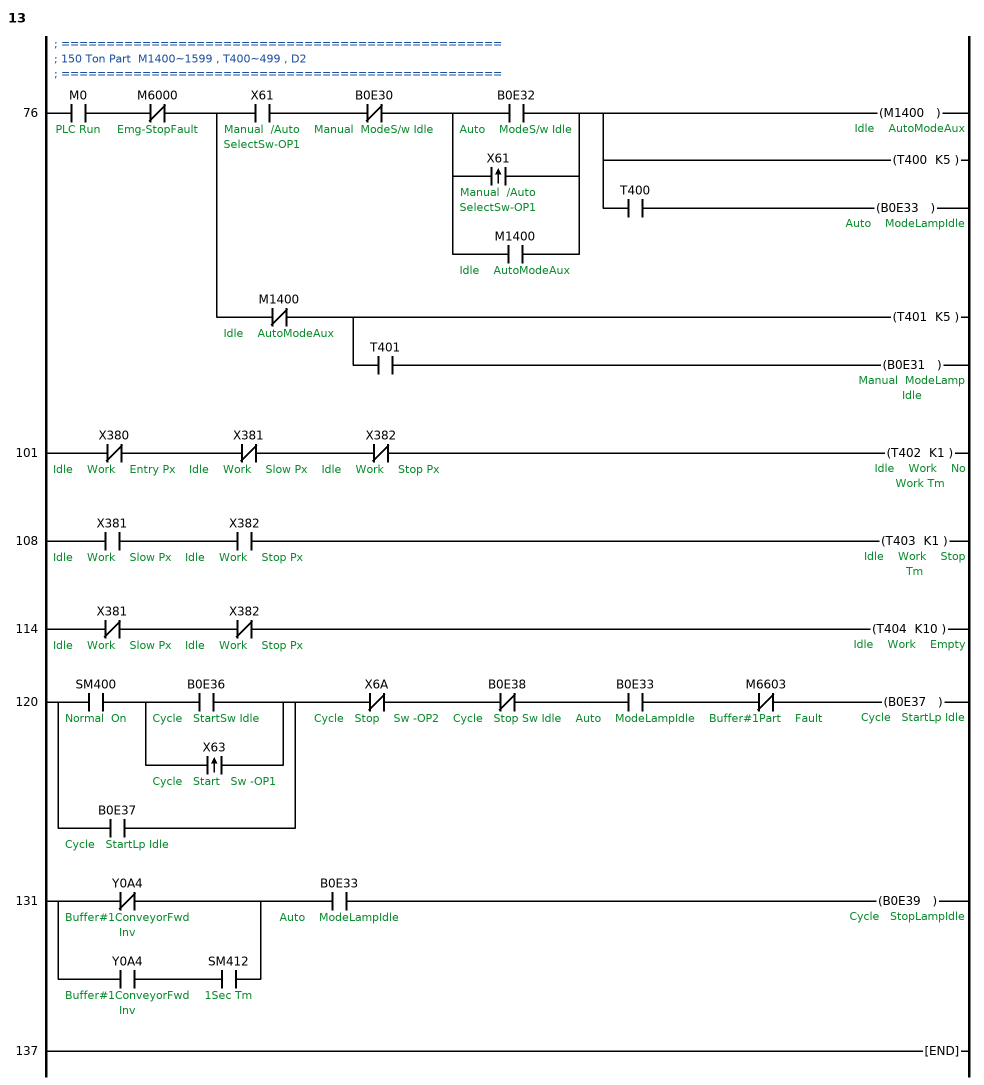
; =================================================
; 150 Ton Part  M1400~1599 , T400~499 , D2
; =================================================
76    LD      M0  ; PLC Run
      ANI     M6000  ; Emg-StopFault
      MPS
      AND     X61  ; Manual  /Auto   SelectSw-OP1
      ANI     B0E30  ; Manual  ModeS/w Idle
      LD      B0E32  ; Auto    ModeS/w Idle
      ORP     X61  ; Manual  /Auto   SelectSw-OP1
      OR      M1400  ; Idle    AutoModeAux
      ANB
      OUT     M1400  ; Idle    AutoModeAux
      OUT     T400 K5
      AND     T400
      OUT     B0E33  ; Auto    ModeLampIdle
      MPP
      ANI     M1400  ; Idle    AutoModeAux
      OUT     T401 K5
      AND     T401
      OUT     B0E31  ; Manual  ModeLampIdle
101   LDI     X380  ; Idle    Work    Entry Px
      ANI     X381  ; Idle    Work    Slow Px
      ANI     X382  ; Idle    Work    Stop Px
      OUT     T402 K1  ; Idle    Work    No Work Tm
108   LD      X381  ; Idle    Work    Slow Px
      AND     X382  ; Idle    Work    Stop Px
      OUT     T403 K1  ; Idle    Work    Stop Tm
114   LDI     X381  ; Idle    Work    Slow Px
      ANI     X382  ; Idle    Work    Stop Px
      OUT     T404 K10  ; Idle    Work    Empty
120   LD      SM400  ; Normal  On
      LD      B0E36  ; Cycle   StartSw Idle
      ORP     X63  ; Cycle   Start   Sw -OP1
      ANB
      OR      B0E37  ; Cycle   StartLp Idle
      ANI     X6A  ; Cycle   Stop    Sw -OP2
      ANI     B0E38  ; Cycle   Stop Sw Idle
      AND     B0E33  ; Auto    ModeLampIdle
      ANI     M6603  ; Buffer#1Part    Fault
      OUT     B0E37  ; Cycle   StartLp Idle
131   LDI     Y0A4  ; Buffer#1ConveyorFwd Inv
      LD      Y0A4  ; Buffer#1ConveyorFwd Inv
      AND     SM412  ; 1Sec Tm
      ORB
      AND     B0E33  ; Auto    ModeLampIdle
      OUT     B0E39  ; Cycle   StopLampIdle
137   END
END_PROGRAM

PROGRAM 14  // Turn Over
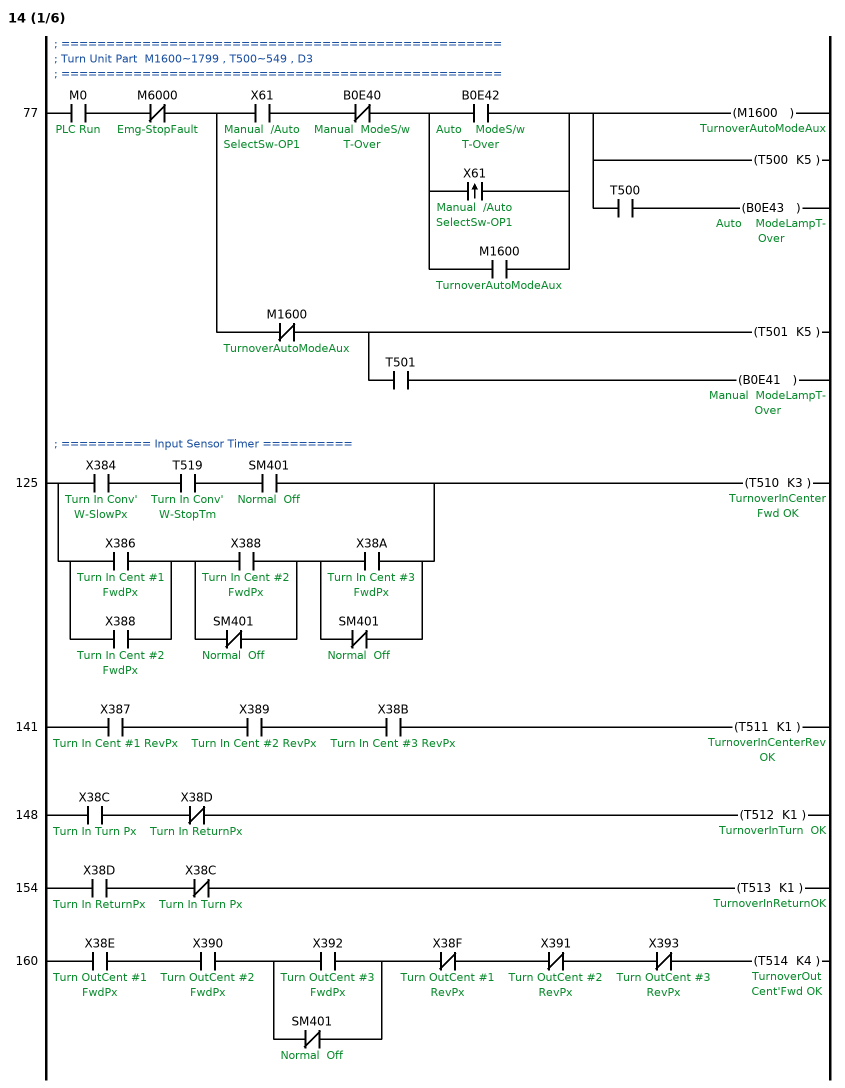
; =================================================
; Turn Unit Part  M1600~1799 , T500~549 , D3
; =================================================
77    LD      M0  ; PLC Run
      ANI     M6000  ; Emg-StopFault
      MPS
      AND     X61  ; Manual  /Auto   SelectSw-OP1
      ANI     B0E40  ; Manual  ModeS/w T-Over
      LD      B0E42  ; Auto    ModeS/w T-Over
      ORP     X61  ; Manual  /Auto   SelectSw-OP1
      OR      M1600  ; TurnoverAutoModeAux
      ANB
      OUT     M1600  ; TurnoverAutoModeAux
      OUT     T500 K5
      AND     T500
      OUT     B0E43  ; Auto    ModeLampT-Over
      MPP
      ANI     M1600  ; TurnoverAutoModeAux
      OUT     T501 K5
      AND     T501
      OUT     B0E41  ; Manual  ModeLampT-Over
; ========== Input Sensor Timer ==========
125   LD      X384  ; Turn In Conv'   W-SlowPx
      AND     T519  ; Turn In Conv'   W-StopTm
      AND     SM401  ; Normal  Off
      LD      X386  ; Turn In Cent #1 FwdPx
      OR      X388  ; Turn In Cent #2 FwdPx
      LD      X388  ; Turn In Cent #2 FwdPx
      ORI     SM401  ; Normal  Off
      ANB
      LD      X38A  ; Turn In Cent #3 FwdPx
      ORI     SM401  ; Normal  Off
      ANB
      ORB
      OUT     T510 K3  ; TurnoverInCenterFwd OK
141   LD      X387  ; Turn In Cent #1 RevPx
      AND     X389  ; Turn In Cent #2 RevPx
      AND     X38B  ; Turn In Cent #3 RevPx
      OUT     T511 K1  ; TurnoverInCenterRev OK
148   LD      X38C  ; Turn In Turn Px
      ANI     X38D  ; Turn In ReturnPx
      OUT     T512 K1  ; TurnoverInTurn  OK
154   LD      X38D  ; Turn In ReturnPx
      ANI     X38C  ; Turn In Turn Px
      OUT     T513 K1  ; TurnoverInReturnOK
160   LD      X38E  ; Turn OutCent #1 FwdPx
      AND     X390  ; Turn OutCent #2 FwdPx
      LD      X392  ; Turn OutCent #3 FwdPx
      ORI     SM401  ; Normal  Off
      ANB
      ANI     X38F  ; Turn OutCent #1 RevPx
      ANI     X391  ; Turn OutCent #2 RevPx
      ANI     X393  ; Turn OutCent #3 RevPx
      OUT     T514 K4  ; TurnoverOutCent'Fwd OK
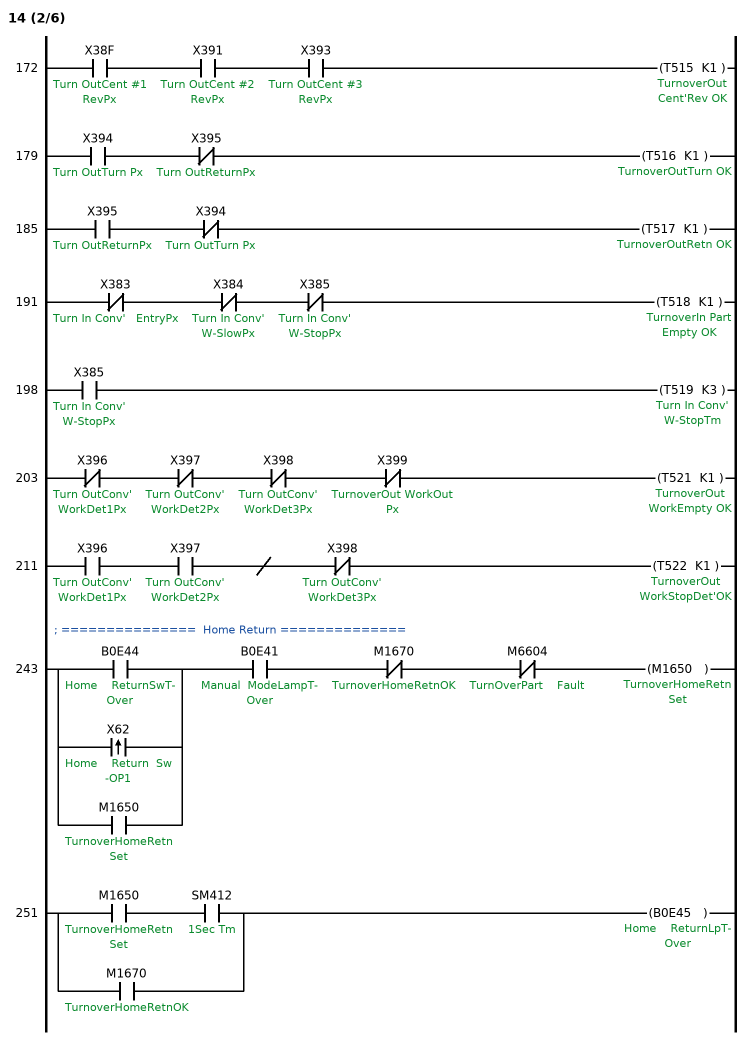
172   LD      X38F  ; Turn OutCent #1 RevPx
      AND     X391  ; Turn OutCent #2 RevPx
      AND     X393  ; Turn OutCent #3 RevPx
      OUT     T515 K1  ; TurnoverOutCent'Rev OK
179   LD      X394  ; Turn OutTurn Px
      ANI     X395  ; Turn OutReturnPx
      OUT     T516 K1  ; TurnoverOutTurn OK
185   LD      X395  ; Turn OutReturnPx
      ANI     X394  ; Turn OutTurn Px
      OUT     T517 K1  ; TurnoverOutRetn OK
191   LDI     X383  ; Turn In Conv'   EntryPx
      ANI     X384  ; Turn In Conv'   W-SlowPx
      ANI     X385  ; Turn In Conv'   W-StopPx
      OUT     T518 K1  ; TurnoverIn Part Empty OK
198   LD      X385  ; Turn In Conv'   W-StopPx
      OUT     T519 K3  ; Turn In Conv'   W-StopTm
203   LDI     X396  ; Turn OutConv'   WorkDet1Px
      ANI     X397  ; Turn OutConv'   WorkDet2Px
      ANI     X398  ; Turn OutConv'   WorkDet3Px
      ANI     X399  ; TurnoverOut WorkOut Px
      OUT     T521 K1  ; TurnoverOut WorkEmpty OK
211   LD      X396  ; Turn OutConv'   WorkDet1Px
      AND     X397  ; Turn OutConv'   WorkDet2Px
      INV
      ANI     X398  ; Turn OutConv'   WorkDet3Px
      OUT     T522 K1  ; TurnoverOut WorkStopDet'OK
; ===============  Home Return ==============
243   LD      B0E44  ; Home    ReturnSwT-Over
      ORP     X62  ; Home    Return  Sw -OP1
      OR      M1650  ; TurnoverHomeRetnSet
      AND     B0E41  ; Manual  ModeLampT-Over
      ANI     M1670  ; TurnoverHomeRetnOK
      ANI     M6604  ; TurnOverPart    Fault
      OUT     M1650  ; TurnoverHomeRetnSet
251   LD      M1650  ; TurnoverHomeRetnSet
      AND     SM412  ; 1Sec Tm
      OR      M1670  ; TurnoverHomeRetnOK
      OUT     B0E45  ; Home    ReturnLpT-Over
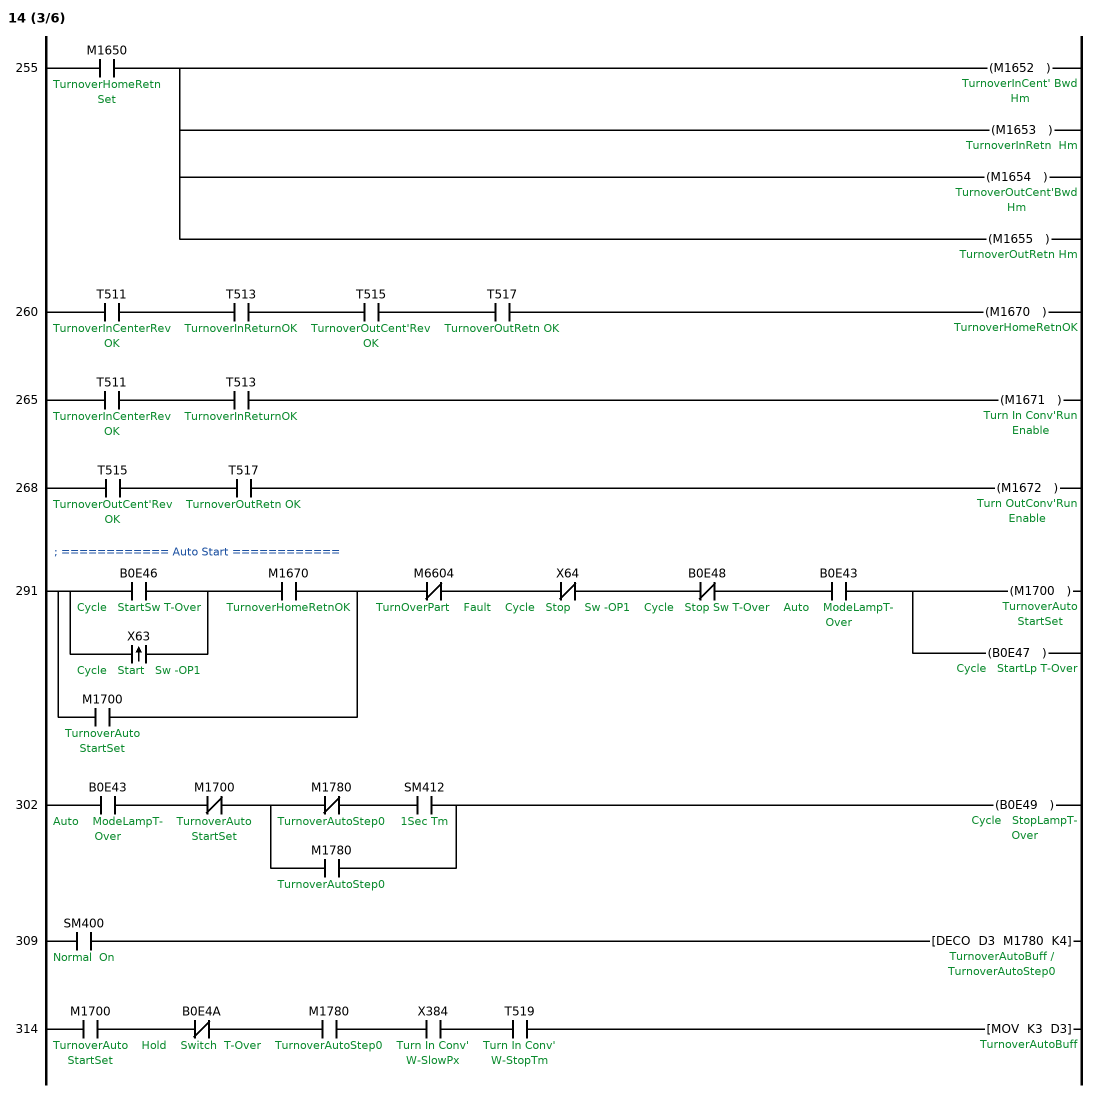
255   LD      M1650  ; TurnoverHomeRetnSet
      OUT     M1652  ; TurnoverInCent' Bwd Hm
      OUT     M1653  ; TurnoverInRetn  Hm
      OUT     M1654  ; TurnoverOutCent'BwdHm
      OUT     M1655  ; TurnoverOutRetn Hm
260   LD      T511  ; TurnoverInCenterRev OK
      AND     T513  ; TurnoverInReturnOK
      AND     T515  ; TurnoverOutCent'Rev OK
      AND     T517  ; TurnoverOutRetn OK
      OUT     M1670  ; TurnoverHomeRetnOK
265   LD      T511  ; TurnoverInCenterRev OK
      AND     T513  ; TurnoverInReturnOK
      OUT     M1671  ; Turn In Conv'RunEnable
268   LD      T515  ; TurnoverOutCent'Rev OK
      AND     T517  ; TurnoverOutRetn OK
      OUT     M1672  ; Turn OutConv'RunEnable
; ============ Auto Start ============
291   LD      B0E46  ; Cycle   StartSw T-Over
      ORP     X63  ; Cycle   Start   Sw -OP1
      AND     M1670  ; TurnoverHomeRetnOK
      OR      M1700  ; TurnoverAuto    StartSet
      ANI     M6604  ; TurnOverPart    Fault
      ANI     X64  ; Cycle   Stop    Sw -OP1
      ANI     B0E48  ; Cycle   Stop Sw T-Over
      AND     B0E43  ; Auto    ModeLampT-Over
      OUT     M1700  ; TurnoverAuto    StartSet
      OUT     B0E47  ; Cycle   StartLp T-Over
302   LD      B0E43  ; Auto    ModeLampT-Over
      ANI     M1700  ; TurnoverAuto    StartSet
      LDI     M1780  ; TurnoverAutoStep0
      AND     SM412  ; 1Sec Tm
      OR      M1780  ; TurnoverAutoStep0
      ANB
      OUT     B0E49  ; Cycle   StopLampT-Over
309   LD      SM400  ; Normal  On
      DECO    D3 M1780 K4  ; TurnoverAutoBuff
314   LD      M1700  ; TurnoverAuto    StartSet
      ANI     B0E4A  ; Hold    Switch  T-Over
      AND     M1780  ; TurnoverAutoStep0
      AND     X384  ; Turn In Conv'   W-SlowPx
      AND     T519  ; Turn In Conv'   W-StopTm
      MOV     K3 D3
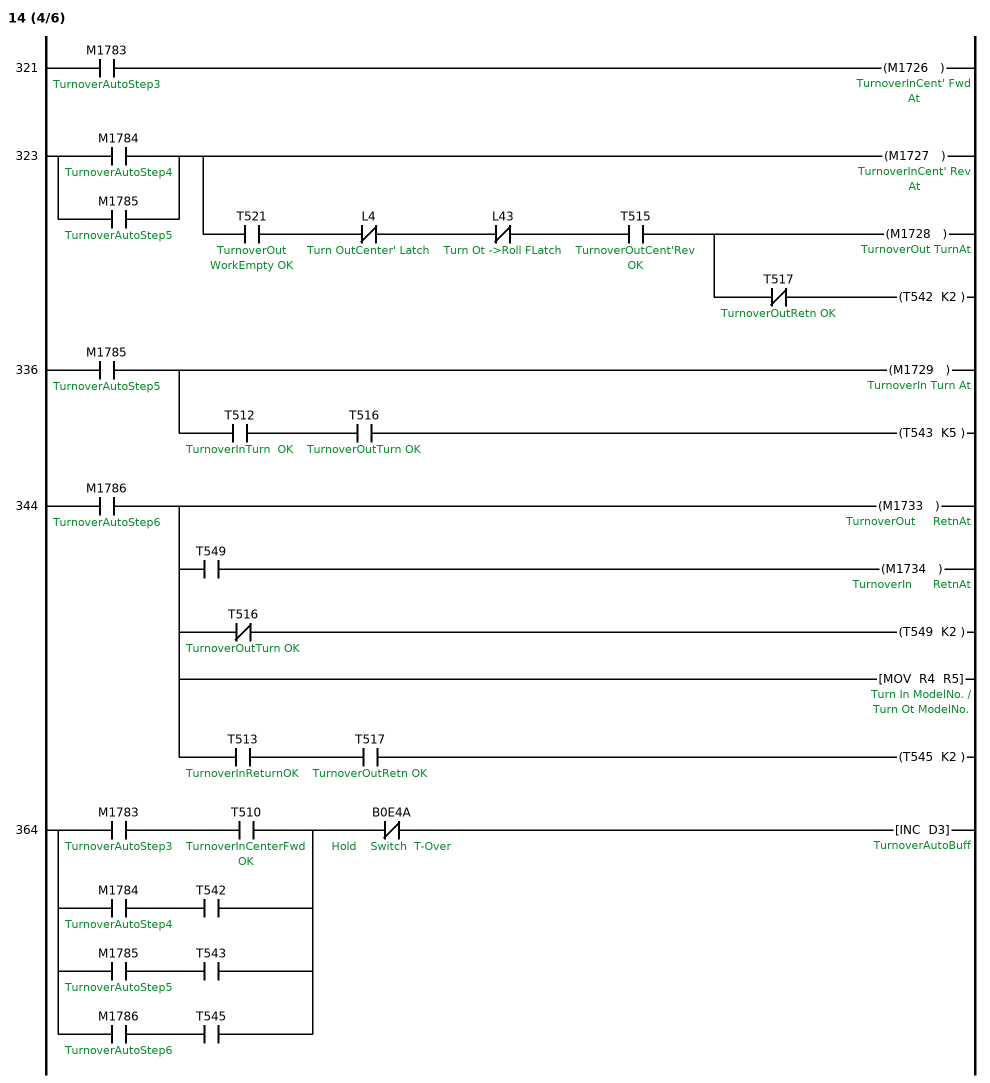
321   LD      M1783  ; TurnoverAutoStep3
      OUT     M1726  ; TurnoverInCent' Fwd At
323   LD      M1784  ; TurnoverAutoStep4
      OR      M1785  ; TurnoverAutoStep5
      OUT     M1727  ; TurnoverInCent' Rev At
      AND     T521  ; TurnoverOut WorkEmpty OK
      ANI     L4  ; Turn OutCenter' Latch
      ANI     L43  ; Turn Ot ->Roll FLatch
      AND     T515  ; TurnoverOutCent'Rev OK
      OUT     M1728  ; TurnoverOut TurnAt
      ANI     T517  ; TurnoverOutRetn OK
      OUT     T542 K2
336   LD      M1785  ; TurnoverAutoStep5
      OUT     M1729  ; TurnoverIn Turn At
      AND     T512  ; TurnoverInTurn  OK
      AND     T516  ; TurnoverOutTurn OK
      OUT     T543 K5
344   LD      M1786  ; TurnoverAutoStep6
      OUT     M1733  ; TurnoverOut     RetnAt
      MPS
      AND     T549
      OUT     M1734  ; TurnoverIn      RetnAt
      MRD
      ANI     T516  ; TurnoverOutTurn OK
      OUT     T549 K2
      MPP
      MOV     R4 R5  ; Turn In ModelNo. / Turn Ot ModelNo.
      AND     T513  ; TurnoverInReturnOK
      AND     T517  ; TurnoverOutRetn OK
      OUT     T545 K2
364   LD      M1783  ; TurnoverAutoStep3
      AND     T510  ; TurnoverInCenterFwd OK
      LD      M1784  ; TurnoverAutoStep4
      AND     T542
      ORB
      LD      M1785  ; TurnoverAutoStep5
      AND     T543
      ORB
      LD      M1786  ; TurnoverAutoStep6
      AND     T545
      ORB
      ANI     B0E4A  ; Hold    Switch  T-Over
      INC     D3
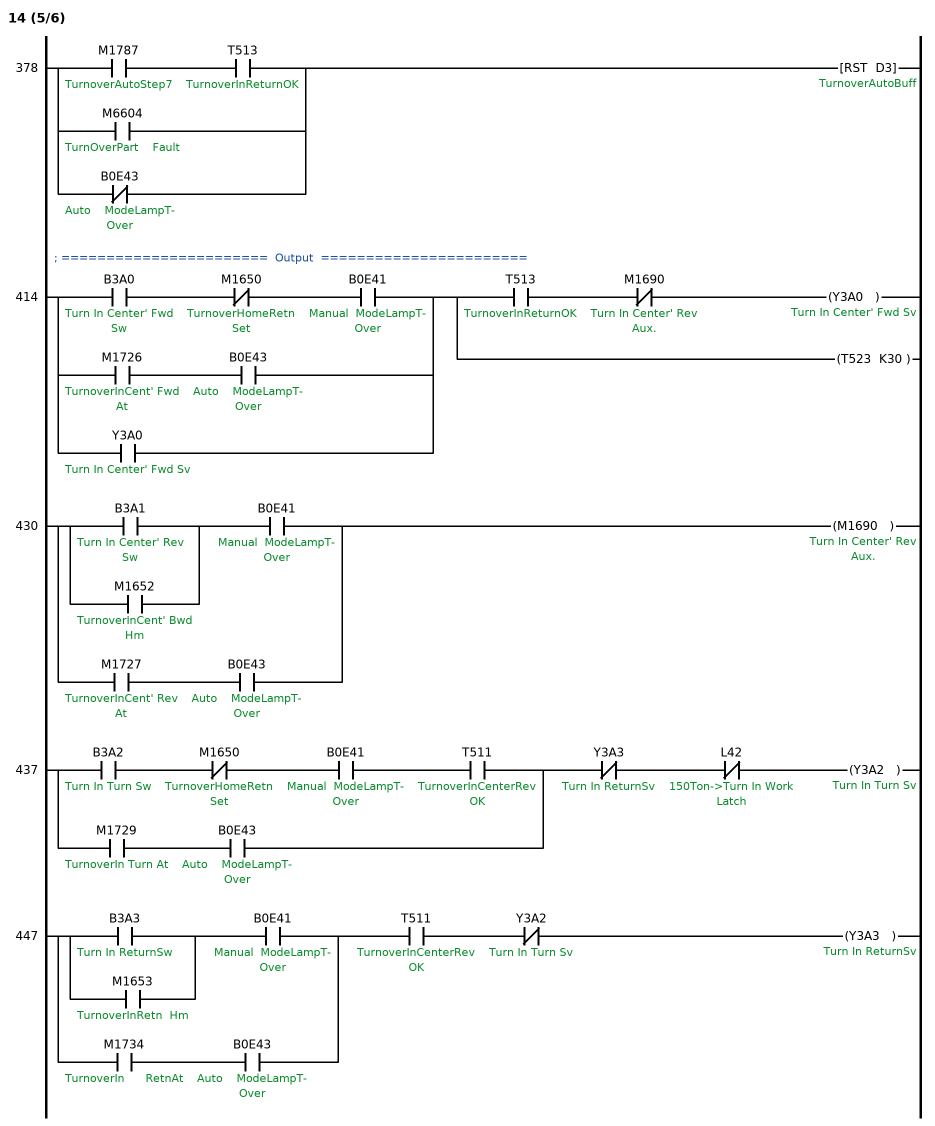
378   LD      M1787  ; TurnoverAutoStep7
      AND     T513  ; TurnoverInReturnOK
      OR      M6604  ; TurnOverPart    Fault
      ORI     B0E43  ; Auto    ModeLampT-Over
      RST     D3  ; TurnoverAutoBuff
; =======================  Output  =======================
414   LD      B3A0  ; Turn In Center' Fwd Sw
      ANI     M1650  ; TurnoverHomeRetnSet
      AND     B0E41  ; Manual  ModeLampT-Over
      LD      M1726  ; TurnoverInCent' Fwd At
      AND     B0E43  ; Auto    ModeLampT-Over
      ORB
      OR      Y3A0  ; Turn In Center' Fwd Sv
      MPS
      AND     T513  ; TurnoverInReturnOK
      ANI     M1690  ; Turn In Center' Rev Aux.
      OUT     Y3A0  ; Turn In Center' Fwd Sv
      MPP
      OUT     T523 K30
430   LD      B3A1  ; Turn In Center' Rev Sw
      OR      M1652  ; TurnoverInCent' Bwd Hm
      AND     B0E41  ; Manual  ModeLampT-Over
      LD      M1727  ; TurnoverInCent' Rev At
      AND     B0E43  ; Auto    ModeLampT-Over
      ORB
      OUT     M1690  ; Turn In Center' Rev Aux.
437   LD      B3A2  ; Turn In Turn Sw
      ANI     M1650  ; TurnoverHomeRetnSet
      AND     B0E41  ; Manual  ModeLampT-Over
      AND     T511  ; TurnoverInCenterRev OK
      LD      M1729  ; TurnoverIn Turn At
      AND     B0E43  ; Auto    ModeLampT-Over
      ORB
      ANI     Y3A3  ; Turn In ReturnSv
      ANI     L42  ; 150Ton->Turn In Work    Latch
      OUT     Y3A2  ; Turn In Turn Sv
447   LD      B3A3  ; Turn In ReturnSw
      OR      M1653  ; TurnoverInRetn  Hm
      AND     B0E41  ; Manual  ModeLampT-Over
      LD      M1734  ; TurnoverIn      RetnAt
      AND     B0E43  ; Auto    ModeLampT-Over
      ORB
      AND     T511  ; TurnoverInCenterRev OK
      ANI     Y3A2  ; Turn In Turn Sv
      OUT     Y3A3  ; Turn In ReturnSv
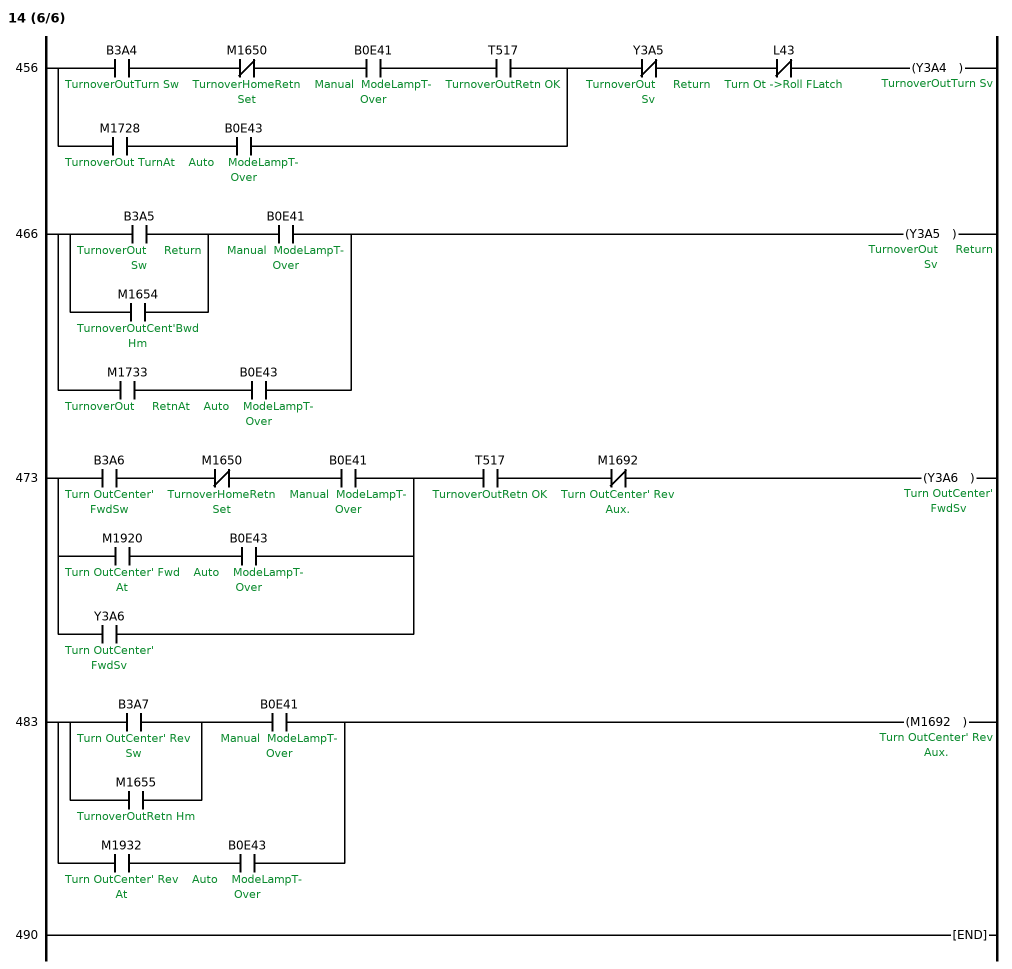
456   LD      B3A4  ; TurnoverOutTurn Sw
      ANI     M1650  ; TurnoverHomeRetnSet
      AND     B0E41  ; Manual  ModeLampT-Over
      AND     T517  ; TurnoverOutRetn OK
      LD      M1728  ; TurnoverOut TurnAt
      AND     B0E43  ; Auto    ModeLampT-Over
      ORB
      ANI     Y3A5  ; TurnoverOut     Return  Sv
      ANI     L43  ; Turn Ot ->Roll FLatch
      OUT     Y3A4  ; TurnoverOutTurn Sv
466   LD      B3A5  ; TurnoverOut     Return  Sw
      OR      M1654  ; TurnoverOutCent'BwdHm
      AND     B0E41  ; Manual  ModeLampT-Over
      LD      M1733  ; TurnoverOut     RetnAt
      AND     B0E43  ; Auto    ModeLampT-Over
      ORB
      OUT     Y3A5  ; TurnoverOut     Return  Sv
473   LD      B3A6  ; Turn OutCenter' FwdSw
      ANI     M1650  ; TurnoverHomeRetnSet
      AND     B0E41  ; Manual  ModeLampT-Over
      LD      M1920  ; Turn OutCenter' Fwd At
      AND     B0E43  ; Auto    ModeLampT-Over
      ORB
      OR      Y3A6  ; Turn OutCenter' FwdSv
      AND     T517  ; TurnoverOutRetn OK
      ANI     M1692  ; Turn OutCenter' Rev Aux.
      OUT     Y3A6  ; Turn OutCenter' FwdSv
483   LD      B3A7  ; Turn OutCenter' Rev Sw
      OR      M1655  ; TurnoverOutRetn Hm
      AND     B0E41  ; Manual  ModeLampT-Over
      LD      M1932  ; Turn OutCenter' Rev At
      AND     B0E43  ; Auto    ModeLampT-Over
      ORB
      OUT     M1692  ; Turn OutCenter' Rev Aux.
490   END
END_PROGRAM

PROGRAM 15  // Roll Forming
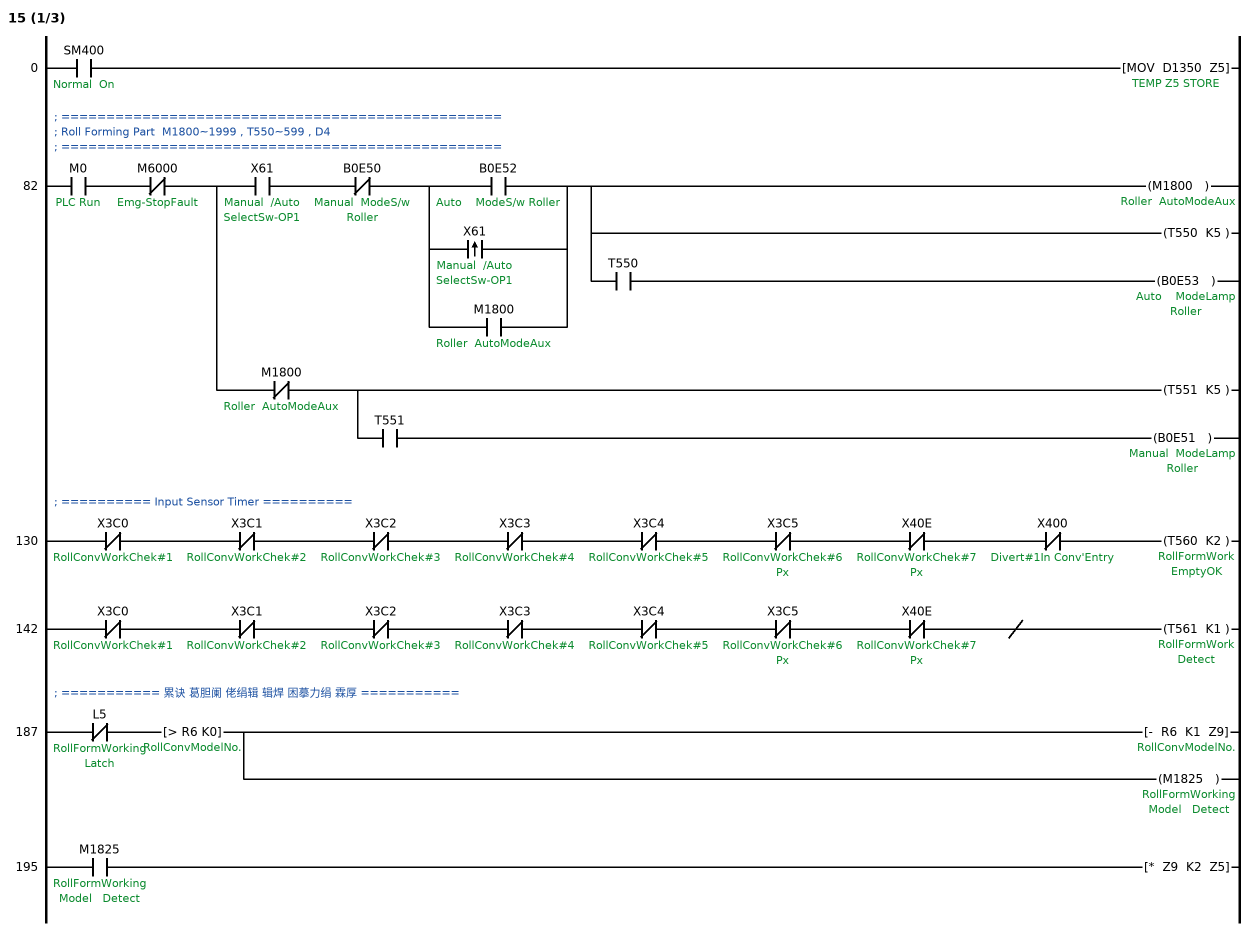
0     LD      SM400  ; Normal  On
      MOV     D1350 Z5  ; TEMP Z5 STORE
; =================================================
; Roll Forming Part  M1800~1999 , T550~599 , D4
; =================================================
82    LD      M0  ; PLC Run
      ANI     M6000  ; Emg-StopFault
      MPS
      AND     X61  ; Manual  /Auto   SelectSw-OP1
      ANI     B0E50  ; Manual  ModeS/w Roller
      LD      B0E52  ; Auto    ModeS/w Roller
      ORP     X61  ; Manual  /Auto   SelectSw-OP1
      OR      M1800  ; Roller  AutoModeAux
      ANB
      OUT     M1800  ; Roller  AutoModeAux
      OUT     T550 K5
      AND     T550
      OUT     B0E53  ; Auto    ModeLampRoller
      MPP
      ANI     M1800  ; Roller  AutoModeAux
      OUT     T551 K5
      AND     T551
      OUT     B0E51  ; Manual  ModeLampRoller
; ========== Input Sensor Timer ==========
130   LDI     X3C0  ; RollConvWorkChek#1
      ANI     X3C1  ; RollConvWorkChek#2
      ANI     X3C2  ; RollConvWorkChek#3
      ANI     X3C3  ; RollConvWorkChek#4
      ANI     X3C4  ; RollConvWorkChek#5
      ANI     X3C5  ; RollConvWorkChek#6 Px
      ANI     X40E  ; RollConvWorkChek#7 Px
      ANI     X400  ; Divert#1In Conv'Entry
      OUT     T560 K2  ; RollFormWork    EmptyOK
142   LDI     X3C0  ; RollConvWorkChek#1
      ANI     X3C1  ; RollConvWorkChek#2
      ANI     X3C2  ; RollConvWorkChek#3
      ANI     X3C3  ; RollConvWorkChek#4
      ANI     X3C4  ; RollConvWorkChek#5
      ANI     X3C5  ; RollConvWorkChek#6 Px
      ANI     X40E  ; RollConvWorkChek#7 Px
      INV
      OUT     T561 K1  ; RollFormWork    Detect
; =========== 작업 모델을 읽어서 서보 위치제어 준비 ===========
187   LDI     L5  ; RollFormWorking Latch
      AND>    R6 K0  ; RollConvModelNo.
      -       R6 K1 Z9
      OUT     M1825  ; RollFormWorking Model   Detect
195   LD      M1825  ; RollFormWorking Model   Detect
      *       Z9 K2 Z5
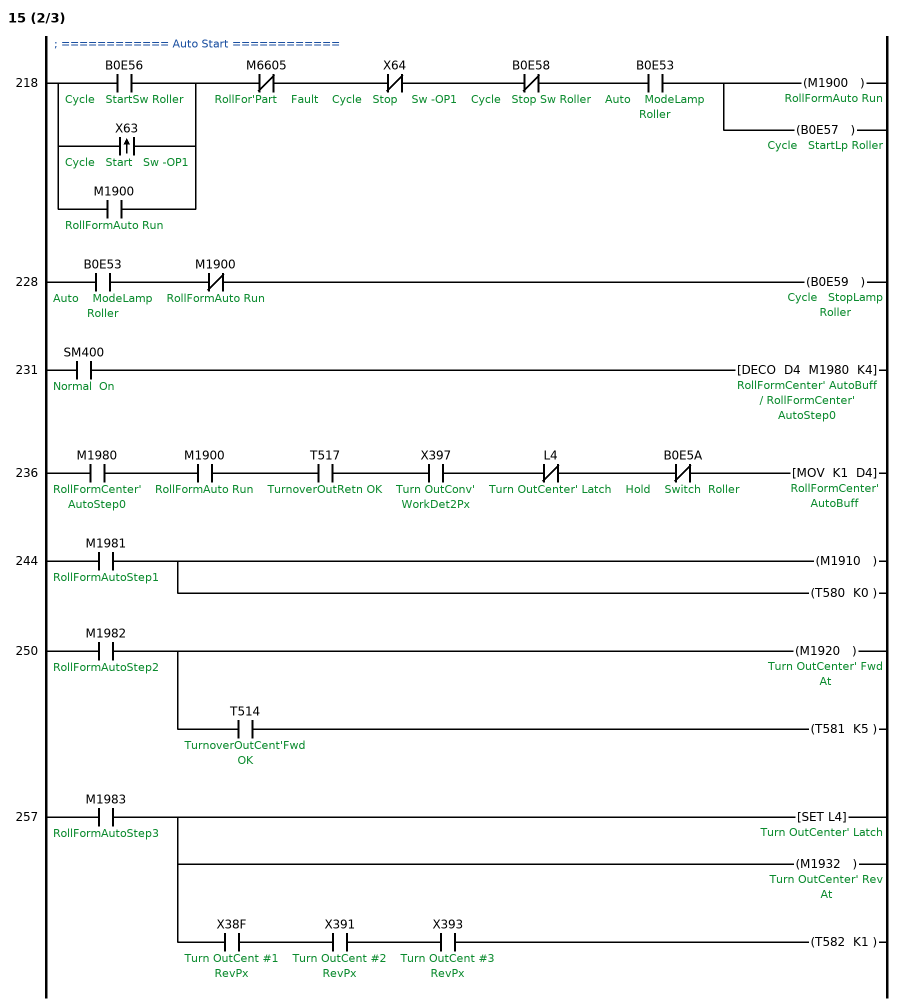
; ============ Auto Start ============
218   LD      B0E56  ; Cycle   StartSw Roller
      ORP     X63  ; Cycle   Start   Sw -OP1
      OR      M1900  ; RollFormAuto Run
      ANI     M6605  ; RollFor'Part    Fault
      ANI     X64  ; Cycle   Stop    Sw -OP1
      ANI     B0E58  ; Cycle   Stop Sw Roller
      AND     B0E53  ; Auto    ModeLampRoller
      OUT     M1900  ; RollFormAuto Run
      OUT     B0E57  ; Cycle   StartLp Roller
228   LD      B0E53  ; Auto    ModeLampRoller
      ANI     M1900  ; RollFormAuto Run
      OUT     B0E59  ; Cycle   StopLampRoller
231   LD      SM400  ; Normal  On
      DECO    D4 M1980 K4  ; RollFormCenter' AutoBuff / RollFormCenter' AutoStep0
236   LD      M1980  ; RollFormCenter' AutoStep0
      AND     M1900  ; RollFormAuto Run
      AND     T517  ; TurnoverOutRetn OK
      AND     X397  ; Turn OutConv'   WorkDet2Px
      ANI     L4  ; Turn OutCenter' Latch
      ANI     B0E5A  ; Hold    Switch  Roller
      MOV     K1 D4
244   LD      M1981  ; RollFormAutoStep1
      OUT     M1910
      OUT     T580 K0
250   LD      M1982  ; RollFormAutoStep2
      OUT     M1920  ; Turn OutCenter' Fwd At
      AND     T514  ; TurnoverOutCent'Fwd OK
      OUT     T581 K5
257   LD      M1983  ; RollFormAutoStep3
      SET     L4  ; Turn OutCenter' Latch
      OUT     M1932  ; Turn OutCenter' Rev At
      AND     X38F  ; Turn OutCent #1 RevPx
      AND     X391  ; Turn OutCent #2 RevPx
      AND     X393  ; Turn OutCent #3 RevPx
      OUT     T582 K1
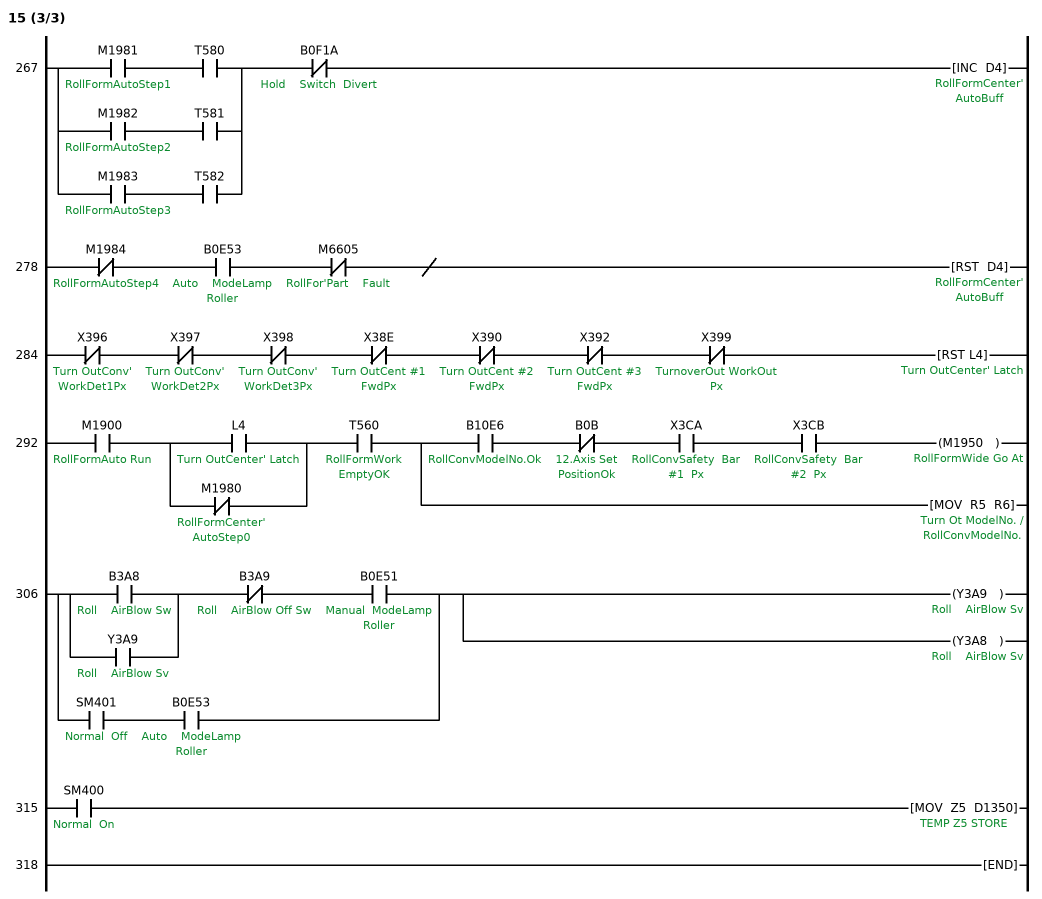
267   LD      M1981  ; RollFormAutoStep1
      AND     T580
      LD      M1982  ; RollFormAutoStep2
      AND     T581
      ORB
      LD      M1983  ; RollFormAutoStep3
      AND     T582
      ORB
      ANI     B0F1A  ; Hold    Switch  Divert
      INC     D4
278   LDI     M1984  ; RollFormAutoStep4
      AND     B0E53  ; Auto    ModeLampRoller
      ANI     M6605  ; RollFor'Part    Fault
      INV
      RST     D4  ; RollFormCenter' AutoBuff
284   LDI     X396  ; Turn OutConv'   WorkDet1Px
      ANI     X397  ; Turn OutConv'   WorkDet2Px
      ANI     X398  ; Turn OutConv'   WorkDet3Px
      ANI     X38E  ; Turn OutCent #1 FwdPx
      ANI     X390  ; Turn OutCent #2 FwdPx
      ANI     X392  ; Turn OutCent #3 FwdPx
      ANI     X399  ; TurnoverOut WorkOut Px
      RST     L4  ; Turn OutCenter' Latch
292   LD      M1900  ; RollFormAuto Run
      LD      L4  ; Turn OutCenter' Latch
      ORI     M1980  ; RollFormCenter' AutoStep0
      ANB
      AND     T560  ; RollFormWork    EmptyOK
      MPS
      AND     B10E6  ; RollConvModelNo.Ok
      ANI     B0B  ; 12.Axis Set     PositionOk
      AND     X3CA  ; RollConvSafety  Bar #1  Px
      AND     X3CB  ; RollConvSafety  Bar #2  Px
      OUT     M1950  ; RollFormWide Go At
      MPP
      MOV     R5 R6  ; Turn Ot ModelNo.
306   LD      B3A8  ; Roll    AirBlow Sw
      OR      Y3A9  ; Roll    AirBlow Sv
      ANI     B3A9  ; Roll    AirBlow Off Sw
      AND     B0E51  ; Manual  ModeLampRoller
      LD      SM401  ; Normal  Off
      AND     B0E53  ; Auto    ModeLampRoller
      ORB
      OUT     Y3A9  ; Roll    AirBlow Sv
      OUT     Y3A8  ; Roll    AirBlow Sv
315   LD      SM400  ; Normal  On
      MOV     Z5 D1350
318   END
END_PROGRAM

PROGRAM 19  // #2 Part Alarm
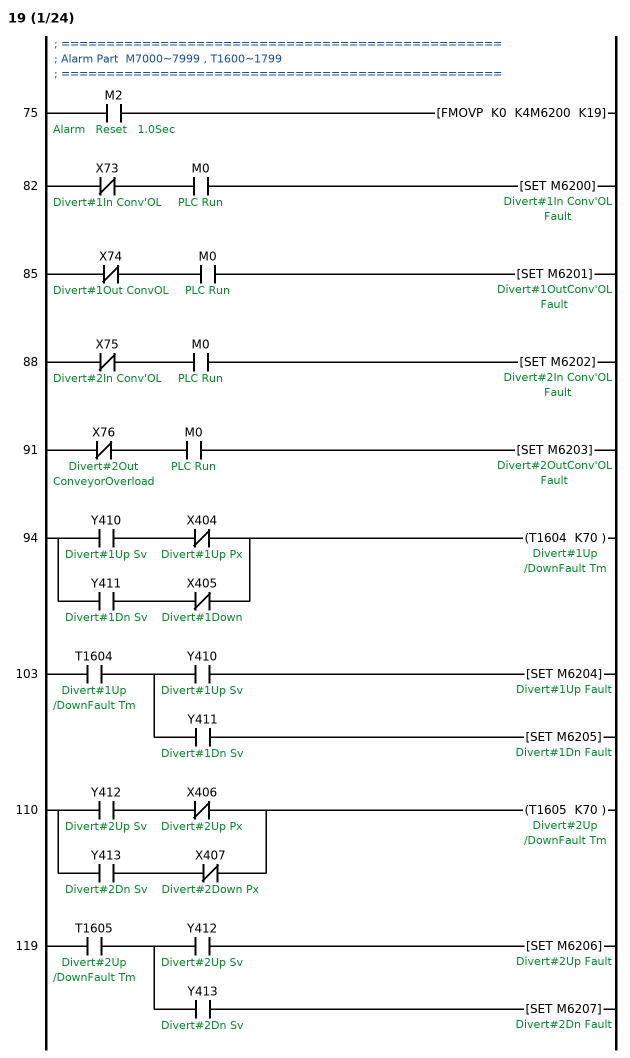
; =================================================
; Alarm Part  M7000~7999 , T1600~1799
; =================================================
75    LD      M2  ; Alarm   Reset   1.0Sec
      FMOVP   K0 K4M6200 K19  ; Divert#1In Conv'OL Fault
82    LDI     X73  ; Divert#1In Conv'OL
      AND     M0  ; PLC Run
      SET     M6200  ; Divert#1In Conv'OL Fault
85    LDI     X74  ; Divert#1Out ConvOL
      AND     M0  ; PLC Run
      SET     M6201  ; Divert#1OutConv'OL Fault
88    LDI     X75  ; Divert#2In Conv'OL
      AND     M0  ; PLC Run
      SET     M6202  ; Divert#2In Conv'OL Fault
91    LDI     X76  ; Divert#2Out     ConveyorOverload
      AND     M0  ; PLC Run
      SET     M6203  ; Divert#2OutConv'OL Fault
94    LD      Y410  ; Divert#1Up Sv
      ANI     X404  ; Divert#1Up Px
      LD      Y411  ; Divert#1Dn Sv
      ANI     X405  ; Divert#1Down
      ORB
      OUT     T1604 K70  ; Divert#1Up /DownFault Tm
103   LD      T1604  ; Divert#1Up /DownFault Tm
      MPS
      AND     Y410  ; Divert#1Up Sv
      SET     M6204  ; Divert#1Up Fault
      MPP
      AND     Y411  ; Divert#1Dn Sv
      SET     M6205  ; Divert#1Dn Fault
110   LD      Y412  ; Divert#2Up Sv
      ANI     X406  ; Divert#2Up Px
      LD      Y413  ; Divert#2Dn Sv
      ANI     X407  ; Divert#2Down Px
      ORB
      OUT     T1605 K70  ; Divert#2Up /DownFault Tm
119   LD      T1605  ; Divert#2Up /DownFault Tm
      MPS
      AND     Y412  ; Divert#2Up Sv
      SET     M6206  ; Divert#2Up Fault
      MPP
      AND     Y413  ; Divert#2Dn Sv
      SET     M6207  ; Divert#2Dn Fault
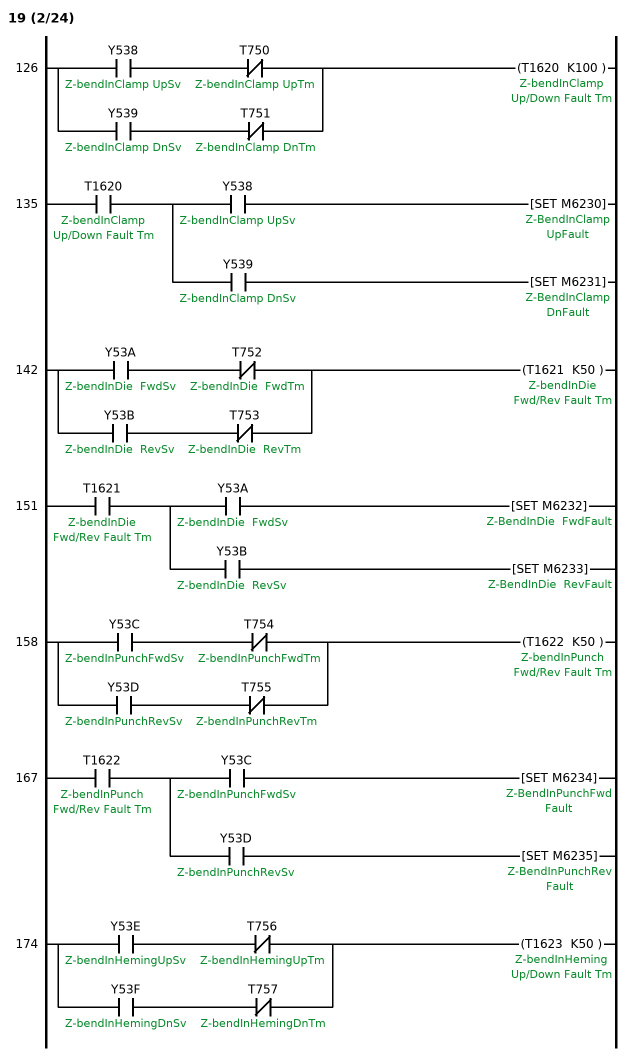
126   LD      Y538  ; Z-bendInClamp UpSv
      ANI     T750  ; Z-bendInClamp UpTm
      LD      Y539  ; Z-bendInClamp DnSv
      ANI     T751  ; Z-bendInClamp DnTm
      ORB
      OUT     T1620 K100  ; Z-bendInClamp   Up/Down Fault Tm
135   LD      T1620  ; Z-bendInClamp   Up/Down Fault Tm
      MPS
      AND     Y538  ; Z-bendInClamp UpSv
      SET     M6230  ; Z-BendInClamp UpFault
      MPP
      AND     Y539  ; Z-bendInClamp DnSv
      SET     M6231  ; Z-BendInClamp DnFault
142   LD      Y53A  ; Z-bendInDie  FwdSv
      ANI     T752  ; Z-bendInDie  FwdTm
      LD      Y53B  ; Z-bendInDie  RevSv
      ANI     T753  ; Z-bendInDie  RevTm
      ORB
      OUT     T1621 K50  ; Z-bendInDie     Fwd/Rev Fault Tm
151   LD      T1621  ; Z-bendInDie     Fwd/Rev Fault Tm
      MPS
      AND     Y53A  ; Z-bendInDie  FwdSv
      SET     M6232  ; Z-BendInDie  FwdFault
      MPP
      AND     Y53B  ; Z-bendInDie  RevSv
      SET     M6233  ; Z-BendInDie  RevFault
158   LD      Y53C  ; Z-bendInPunchFwdSv
      ANI     T754  ; Z-bendInPunchFwdTm
      LD      Y53D  ; Z-bendInPunchRevSv
      ANI     T755  ; Z-bendInPunchRevTm
      ORB
      OUT     T1622 K50  ; Z-bendInPunch   Fwd/Rev Fault Tm
167   LD      T1622  ; Z-bendInPunch   Fwd/Rev Fault Tm
      MPS
      AND     Y53C  ; Z-bendInPunchFwdSv
      SET     M6234  ; Z-BendInPunchFwdFault
      MPP
      AND     Y53D  ; Z-bendInPunchRevSv
      SET     M6235  ; Z-BendInPunchRevFault
174   LD      Y53E  ; Z-bendInHemingUpSv
      ANI     T756  ; Z-bendInHemingUpTm
      LD      Y53F  ; Z-bendInHemingDnSv
      ANI     T757  ; Z-bendInHemingDnTm
      ORB
      OUT     T1623 K50  ; Z-bendInHeming  Up/Down Fault Tm
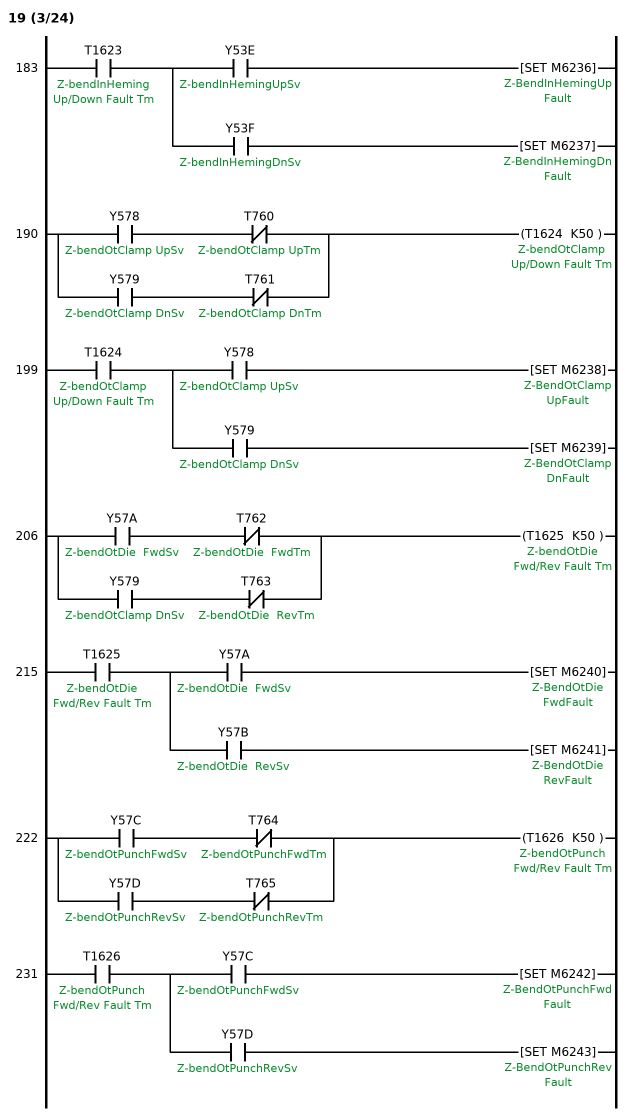
183   LD      T1623  ; Z-bendInHeming  Up/Down Fault Tm
      MPS
      AND     Y53E  ; Z-bendInHemingUpSv
      SET     M6236  ; Z-BendInHemingUpFault
      MPP
      AND     Y53F  ; Z-bendInHemingDnSv
      SET     M6237  ; Z-BendInHemingDnFault
190   LD      Y578  ; Z-bendOtClamp UpSv
      ANI     T760  ; Z-bendOtClamp UpTm
      LD      Y579  ; Z-bendOtClamp DnSv
      ANI     T761  ; Z-bendOtClamp DnTm
      ORB
      OUT     T1624 K50  ; Z-bendOtClamp   Up/Down Fault Tm
199   LD      T1624  ; Z-bendOtClamp   Up/Down Fault Tm
      MPS
      AND     Y578  ; Z-bendOtClamp UpSv
      SET     M6238  ; Z-BendOtClamp UpFault
      MPP
      AND     Y579  ; Z-bendOtClamp DnSv
      SET     M6239  ; Z-BendOtClamp DnFault
206   LD      Y57A  ; Z-bendOtDie  FwdSv
      ANI     T762  ; Z-bendOtDie  FwdTm
      LD      Y579  ; Z-bendOtClamp DnSv
      ANI     T763  ; Z-bendOtDie  RevTm
      ORB
      OUT     T1625 K50  ; Z-bendOtDie     Fwd/Rev Fault Tm
215   LD      T1625  ; Z-bendOtDie     Fwd/Rev Fault Tm
      MPS
      AND     Y57A  ; Z-bendOtDie  FwdSv
      SET     M6240  ; Z-BendOtDie  FwdFault
      MPP
      AND     Y57B  ; Z-bendOtDie  RevSv
      SET     M6241  ; Z-BendOtDie  RevFault
222   LD      Y57C  ; Z-bendOtPunchFwdSv
      ANI     T764  ; Z-bendOtPunchFwdTm
      LD      Y57D  ; Z-bendOtPunchRevSv
      ANI     T765  ; Z-bendOtPunchRevTm
      ORB
      OUT     T1626 K50  ; Z-bendOtPunch   Fwd/Rev Fault Tm
231   LD      T1626  ; Z-bendOtPunch   Fwd/Rev Fault Tm
      MPS
      AND     Y57C  ; Z-bendOtPunchFwdSv
      SET     M6242  ; Z-BendOtPunchFwdFault
      MPP
      AND     Y57D  ; Z-bendOtPunchRevSv
      SET     M6243  ; Z-BendOtPunchRevFault
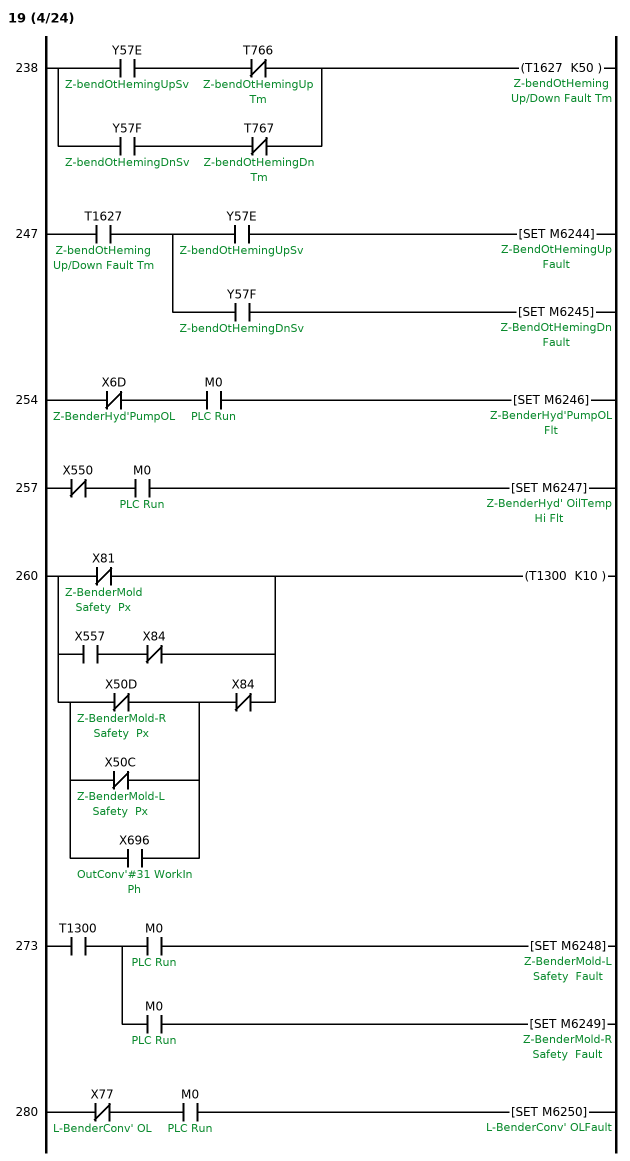
238   LD      Y57E  ; Z-bendOtHemingUpSv
      ANI     T766  ; Z-bendOtHemingUpTm
      LD      Y57F  ; Z-bendOtHemingDnSv
      ANI     T767  ; Z-bendOtHemingDnTm
      ORB
      OUT     T1627 K50  ; Z-bendOtHeming  Up/Down Fault Tm
247   LD      T1627  ; Z-bendOtHeming  Up/Down Fault Tm
      MPS
      AND     Y57E  ; Z-bendOtHemingUpSv
      SET     M6244  ; Z-BendOtHemingUpFault
      MPP
      AND     Y57F  ; Z-bendOtHemingDnSv
      SET     M6245  ; Z-BendOtHemingDnFault
254   LDI     X6D  ; Z-BenderHyd'PumpOL
      AND     M0  ; PLC Run
      SET     M6246  ; Z-BenderHyd'PumpOL Flt
257   LDI     X550
      AND     M0  ; PLC Run
      SET     M6247  ; Z-BenderHyd' OilTemp Hi Flt
260   LDI     X81  ; Z-BenderMold    Safety  Px
      LD      X557
      ANI     X84
      ORB
      LDI     X50D  ; Z-BenderMold-R  Safety  Px
      ORI     X50C  ; Z-BenderMold-L  Safety  Px
      OR      X696  ; OutConv'#31 WorkIn  Ph
      ANI     X84
      ORB
      OUT     T1300 K10
273   LD      T1300
      MPS
      AND     M0  ; PLC Run
      SET     M6248  ; Z-BenderMold-L  Safety  Fault
      MPP
      AND     M0  ; PLC Run
      SET     M6249  ; Z-BenderMold-R  Safety  Fault
280   LDI     X77  ; L-BenderConv' OL
      AND     M0  ; PLC Run
      SET     M6250  ; L-BenderConv' OLFault
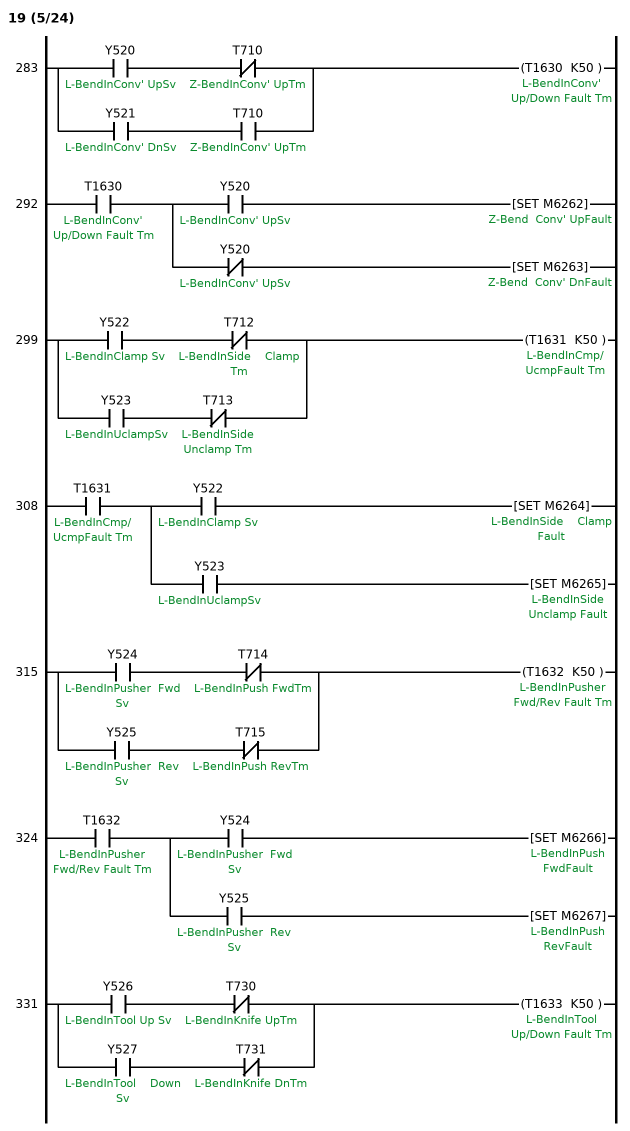
283   LD      Y520  ; L-BendInConv' UpSv
      ANI     T710  ; Z-BendInConv' UpTm
      LD      Y521  ; L-BendInConv' DnSv
      AND     T710  ; Z-BendInConv' UpTm
      ORB
      OUT     T1630 K50  ; L-BendInConv'   Up/Down Fault Tm
292   LD      T1630  ; L-BendInConv'   Up/Down Fault Tm
      MPS
      AND     Y520  ; L-BendInConv' UpSv
      SET     M6262  ; Z-Bend  Conv' UpFault
      MPP
      ANI     Y520  ; L-BendInConv' UpSv
      SET     M6263  ; Z-Bend  Conv' DnFault
299   LD      Y522  ; L-BendInClamp Sv
      ANI     T712  ; L-BendInSide    Clamp Tm
      LD      Y523  ; L-BendInUclampSv
      ANI     T713  ; L-BendInSide    Unclamp Tm
      ORB
      OUT     T1631 K50  ; L-BendInCmp/UcmpFault Tm
308   LD      T1631  ; L-BendInCmp/UcmpFault Tm
      MPS
      AND     Y522  ; L-BendInClamp Sv
      SET     M6264  ; L-BendInSide    Clamp   Fault
      MPP
      AND     Y523  ; L-BendInUclampSv
      SET     M6265  ; L-BendInSide    Unclamp Fault
315   LD      Y524  ; L-BendInPusher  Fwd Sv
      ANI     T714  ; L-BendInPush FwdTm
      LD      Y525  ; L-BendInPusher  Rev Sv
      ANI     T715  ; L-BendInPush RevTm
      ORB
      OUT     T1632 K50  ; L-BendInPusher  Fwd/Rev Fault Tm
324   LD      T1632  ; L-BendInPusher  Fwd/Rev Fault Tm
      MPS
      AND     Y524  ; L-BendInPusher  Fwd Sv
      SET     M6266  ; L-BendInPush    FwdFault
      MPP
      AND     Y525  ; L-BendInPusher  Rev Sv
      SET     M6267  ; L-BendInPush    RevFault
331   LD      Y526  ; L-BendInTool Up Sv
      ANI     T730  ; L-BendInKnife UpTm
      LD      Y527  ; L-BendInTool    Down Sv
      ANI     T731  ; L-BendInKnife DnTm
      ORB
      OUT     T1633 K50  ; L-BendInTool    Up/Down Fault Tm
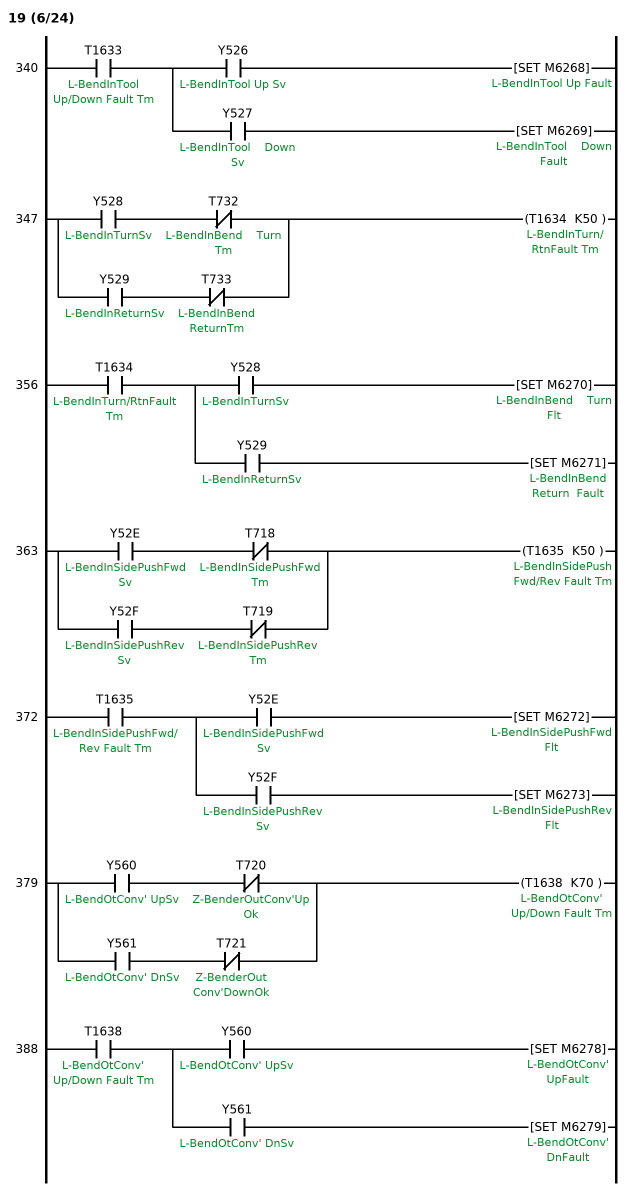
340   LD      T1633  ; L-BendInTool    Up/Down Fault Tm
      MPS
      AND     Y526  ; L-BendInTool Up Sv
      SET     M6268  ; L-BendInTool Up Fault
      MPP
      AND     Y527  ; L-BendInTool    Down Sv
      SET     M6269  ; L-BendInTool    Down    Fault
347   LD      Y528  ; L-BendInTurnSv
      ANI     T732  ; L-BendInBend    Turn Tm
      LD      Y529  ; L-BendInReturnSv
      ANI     T733  ; L-BendInBend    ReturnTm
      ORB
      OUT     T1634 K50  ; L-BendInTurn/RtnFault Tm
356   LD      T1634  ; L-BendInTurn/RtnFault Tm
      MPS
      AND     Y528  ; L-BendInTurnSv
      SET     M6270  ; L-BendInBend    Turn Flt
      MPP
      AND     Y529  ; L-BendInReturnSv
      SET     M6271  ; L-BendInBend    Return  Fault
363   LD      Y52E  ; L-BendInSidePushFwd Sv
      ANI     T718  ; L-BendInSidePushFwd Tm
      LD      Y52F  ; L-BendInSidePushRevSv
      ANI     T719  ; L-BendInSidePushRev Tm
      ORB
      OUT     T1635 K50  ; L-BendInSidePushFwd/Rev Fault Tm
372   LD      T1635  ; L-BendInSidePushFwd/Rev Fault Tm
      MPS
      AND     Y52E  ; L-BendInSidePushFwd Sv
      SET     M6272  ; L-BendInSidePushFwd Flt
      MPP
      AND     Y52F  ; L-BendInSidePushRevSv
      SET     M6273  ; L-BendInSidePushRev Flt
379   LD      Y560  ; L-BendOtConv' UpSv
      ANI     T720  ; Z-BenderOutConv'Up Ok
      LD      Y561  ; L-BendOtConv' DnSv
      ANI     T721  ; Z-BenderOutConv'DownOk
      ORB
      OUT     T1638 K70  ; L-BendOtConv'   Up/Down Fault Tm
388   LD      T1638  ; L-BendOtConv'   Up/Down Fault Tm
      MPS
      AND     Y560  ; L-BendOtConv' UpSv
      SET     M6278  ; L-BendOtConv' UpFault
      MPP
      AND     Y561  ; L-BendOtConv' DnSv
      SET     M6279  ; L-BendOtConv' DnFault
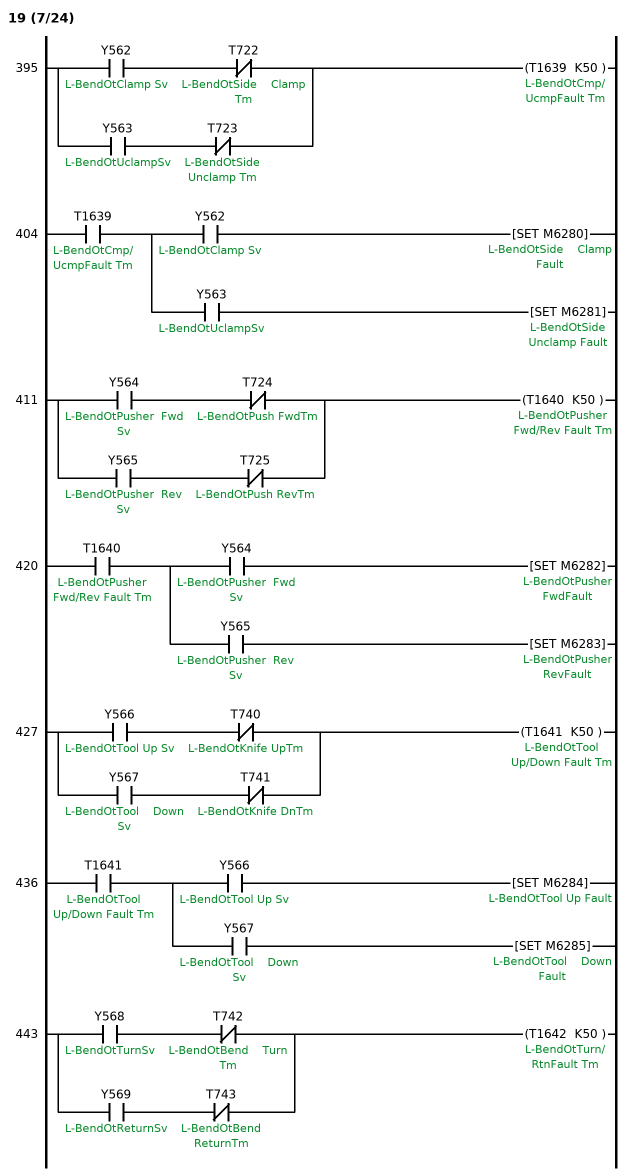
395   LD      Y562  ; L-BendOtClamp Sv
      ANI     T722  ; L-BendOtSide    Clamp Tm
      LD      Y563  ; L-BendOtUclampSv
      ANI     T723  ; L-BendOtSide    Unclamp Tm
      ORB
      OUT     T1639 K50  ; L-BendOtCmp/UcmpFault Tm
404   LD      T1639  ; L-BendOtCmp/UcmpFault Tm
      MPS
      AND     Y562  ; L-BendOtClamp Sv
      SET     M6280  ; L-BendOtSide    Clamp   Fault
      MPP
      AND     Y563  ; L-BendOtUclampSv
      SET     M6281  ; L-BendOtSide    Unclamp Fault
411   LD      Y564  ; L-BendOtPusher  Fwd Sv
      ANI     T724  ; L-BendOtPush FwdTm
      LD      Y565  ; L-BendOtPusher  Rev Sv
      ANI     T725  ; L-BendOtPush RevTm
      ORB
      OUT     T1640 K50  ; L-BendOtPusher  Fwd/Rev Fault Tm
420   LD      T1640  ; L-BendOtPusher  Fwd/Rev Fault Tm
      MPS
      AND     Y564  ; L-BendOtPusher  Fwd Sv
      SET     M6282  ; L-BendOtPusher  FwdFault
      MPP
      AND     Y565  ; L-BendOtPusher  Rev Sv
      SET     M6283  ; L-BendOtPusher  RevFault
427   LD      Y566  ; L-BendOtTool Up Sv
      ANI     T740  ; L-BendOtKnife UpTm
      LD      Y567  ; L-BendOtTool    Down Sv
      ANI     T741  ; L-BendOtKnife DnTm
      ORB
      OUT     T1641 K50  ; L-BendOtTool    Up/Down Fault Tm
436   LD      T1641  ; L-BendOtTool    Up/Down Fault Tm
      MPS
      AND     Y566  ; L-BendOtTool Up Sv
      SET     M6284  ; L-BendOtTool Up Fault
      MPP
      AND     Y567  ; L-BendOtTool    Down Sv
      SET     M6285  ; L-BendOtTool    Down    Fault
443   LD      Y568  ; L-BendOtTurnSv
      ANI     T742  ; L-BendOtBend    Turn Tm
      LD      Y569  ; L-BendOtReturnSv
      ANI     T743  ; L-BendOtBend    ReturnTm
      ORB
      OUT     T1642 K50  ; L-BendOtTurn/RtnFault Tm
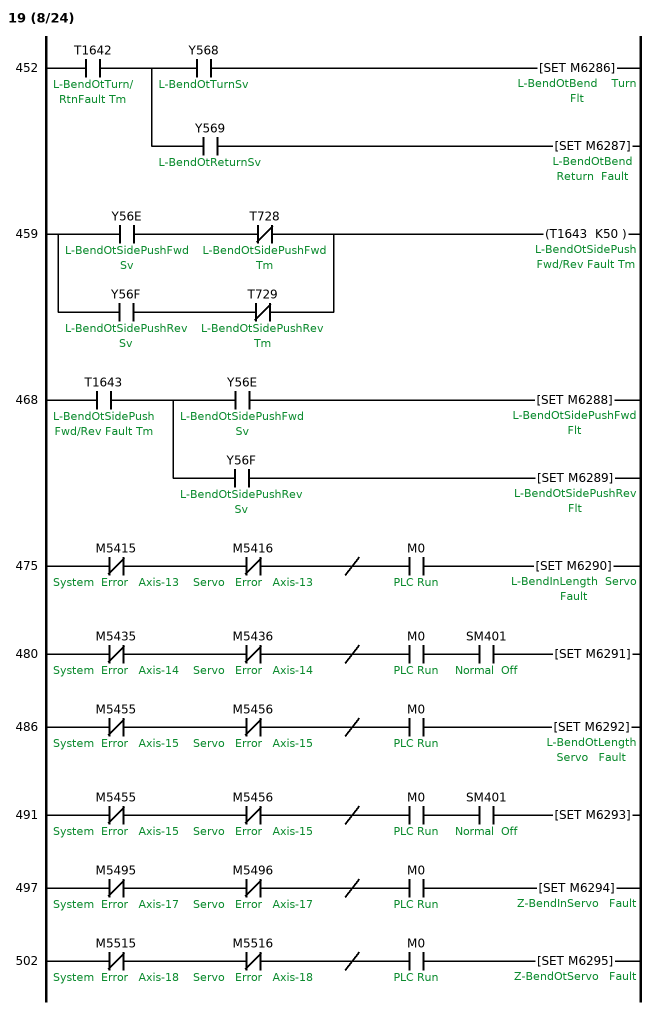
452   LD      T1642  ; L-BendOtTurn/RtnFault Tm
      MPS
      AND     Y568  ; L-BendOtTurnSv
      SET     M6286  ; L-BendOtBend    Turn Flt
      MPP
      AND     Y569  ; L-BendOtReturnSv
      SET     M6287  ; L-BendOtBend    Return  Fault
459   LD      Y56E  ; L-BendOtSidePushFwd Sv
      ANI     T728  ; L-BendOtSidePushFwd Tm
      LD      Y56F  ; L-BendOtSidePushRev Sv
      ANI     T729  ; L-BendOtSidePushRev Tm
      ORB
      OUT     T1643 K50  ; L-BendOtSidePushFwd/Rev Fault Tm
468   LD      T1643  ; L-BendOtSidePushFwd/Rev Fault Tm
      MPS
      AND     Y56E  ; L-BendOtSidePushFwd Sv
      SET     M6288  ; L-BendOtSidePushFwd Flt
      MPP
      AND     Y56F  ; L-BendOtSidePushRev Sv
      SET     M6289  ; L-BendOtSidePushRev Flt
475   LDI     M5415  ; System  Error   Axis-13
      ANI     M5416  ; Servo   Error   Axis-13
      INV
      AND     M0  ; PLC Run
      SET     M6290  ; L-BendInLength  Servo   Fault
480   LDI     M5435  ; System  Error   Axis-14
      ANI     M5436  ; Servo   Error   Axis-14
      INV
      AND     M0  ; PLC Run
      AND     SM401  ; Normal  Off
      SET     M6291
486   LDI     M5455  ; System  Error   Axis-15
      ANI     M5456  ; Servo   Error   Axis-15
      INV
      AND     M0  ; PLC Run
      SET     M6292  ; L-BendOtLength  Servo   Fault
491   LDI     M5455  ; System  Error   Axis-15
      ANI     M5456  ; Servo   Error   Axis-15
      INV
      AND     M0  ; PLC Run
      AND     SM401  ; Normal  Off
      SET     M6293
497   LDI     M5495  ; System  Error   Axis-17
      ANI     M5496  ; Servo   Error   Axis-17
      INV
      AND     M0  ; PLC Run
      SET     M6294  ; Z-BendInServo   Fault
502   LDI     M5515  ; System  Error   Axis-18
      ANI     M5516  ; Servo   Error   Axis-18
      INV
      AND     M0  ; PLC Run
      SET     M6295  ; Z-BendOtServo   Fault
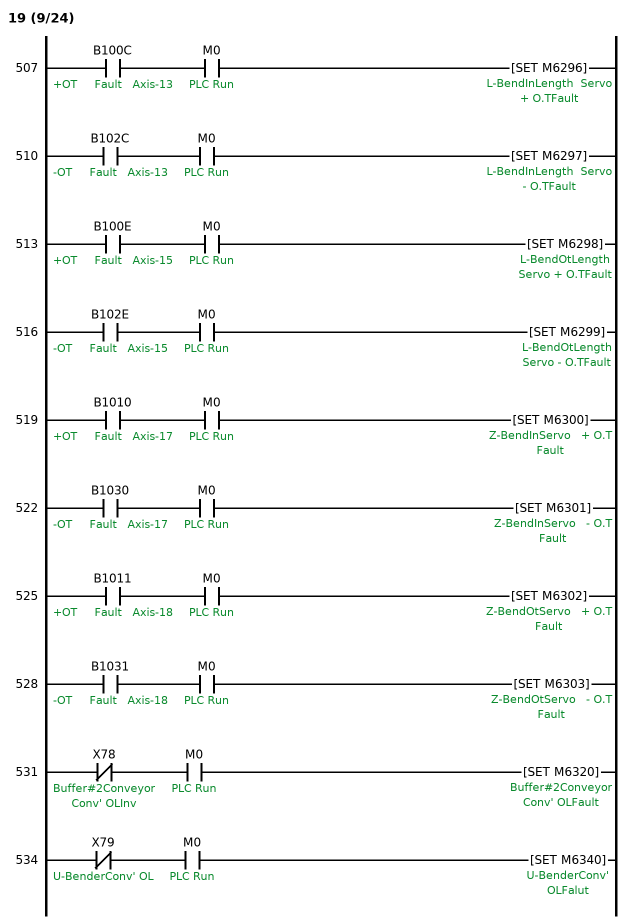
507   LD      B100C  ; +OT     Fault   Axis-13
      AND     M0  ; PLC Run
      SET     M6296  ; L-BendInLength  Servo + O.TFault
510   LD      B102C  ; -OT     Fault   Axis-13
      AND     M0  ; PLC Run
      SET     M6297  ; L-BendInLength  Servo - O.TFault
513   LD      B100E  ; +OT     Fault   Axis-15
      AND     M0  ; PLC Run
      SET     M6298  ; L-BendOtLength  Servo + O.TFault
516   LD      B102E  ; -OT     Fault   Axis-15
      AND     M0  ; PLC Run
      SET     M6299  ; L-BendOtLength  Servo - O.TFault
519   LD      B1010  ; +OT     Fault   Axis-17
      AND     M0  ; PLC Run
      SET     M6300  ; Z-BendInServo   + O.T   Fault
522   LD      B1030  ; -OT     Fault   Axis-17
      AND     M0  ; PLC Run
      SET     M6301  ; Z-BendInServo   - O.T   Fault
525   LD      B1011  ; +OT     Fault   Axis-18
      AND     M0  ; PLC Run
      SET     M6302  ; Z-BendOtServo   + O.T   Fault
528   LD      B1031  ; -OT     Fault   Axis-18
      AND     M0  ; PLC Run
      SET     M6303  ; Z-BendOtServo   - O.T   Fault
531   LDI     X78  ; Buffer#2ConveyorConv' OLInv
      AND     M0  ; PLC Run
      SET     M6320  ; Buffer#2ConveyorConv' OLFault
534   LDI     X79  ; U-BenderConv' OL
      AND     M0  ; PLC Run
      SET     M6340  ; U-BenderConv' OLFalut
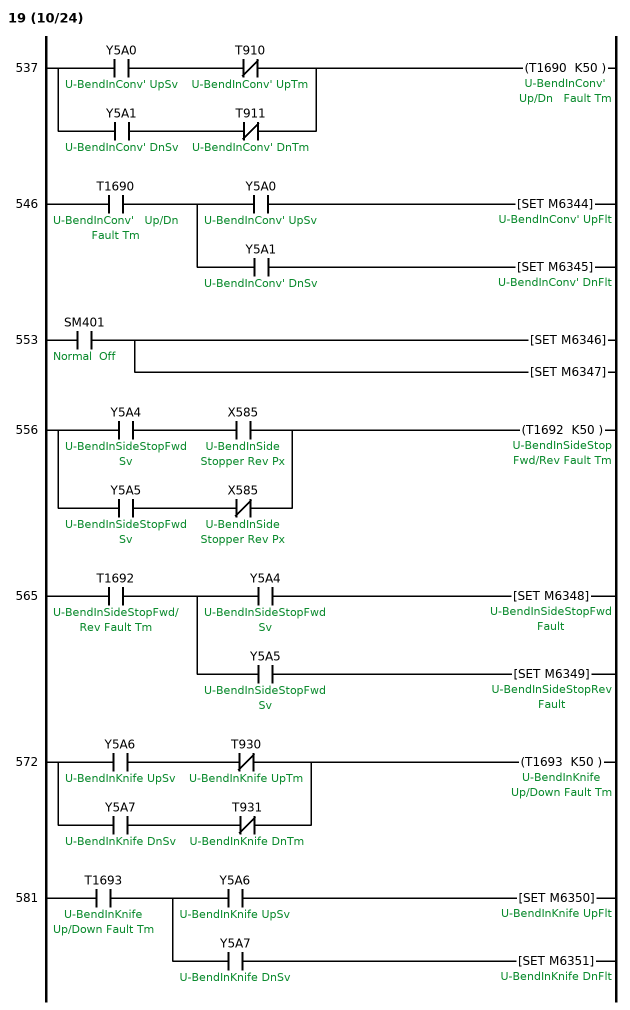
537   LD      Y5A0  ; U-BendInConv' UpSv
      ANI     T910  ; U-BendInConv' UpTm
      LD      Y5A1  ; U-BendInConv' DnSv
      ANI     T911  ; U-BendInConv' DnTm
      ORB
      OUT     T1690 K50  ; U-BendInConv'   Up/Dn   Fault Tm
546   LD      T1690  ; U-BendInConv'   Up/Dn   Fault Tm
      MPS
      AND     Y5A0  ; U-BendInConv' UpSv
      SET     M6344  ; U-BendInConv' UpFlt
      MPP
      AND     Y5A1  ; U-BendInConv' DnSv
      SET     M6345  ; U-BendInConv' DnFlt
553   LD      SM401  ; Normal  Off
      SET     M6346
      SET     M6347
556   LD      Y5A4  ; U-BendInSideStopFwd     Sv
      AND     X585  ; U-BendInSide    Stopper Rev Px
      LD      Y5A5  ; U-BendInSideStopFwd     Sv
      ANI     X585  ; U-BendInSide    Stopper Rev Px
      ORB
      OUT     T1692 K50  ; U-BendInSideStopFwd/Rev Fault Tm
565   LD      T1692  ; U-BendInSideStopFwd/Rev Fault Tm
      MPS
      AND     Y5A4  ; U-BendInSideStopFwd     Sv
      SET     M6348  ; U-BendInSideStopFwd     Fault
      MPP
      AND     Y5A5  ; U-BendInSideStopFwd     Sv
      SET     M6349  ; U-BendInSideStopRev     Fault
572   LD      Y5A6  ; U-BendInKnife UpSv
      ANI     T930  ; U-BendInKnife UpTm
      LD      Y5A7  ; U-BendInKnife DnSv
      ANI     T931  ; U-BendInKnife DnTm
      ORB
      OUT     T1693 K50  ; U-BendInKnife   Up/Down Fault Tm
581   LD      T1693  ; U-BendInKnife   Up/Down Fault Tm
      MPS
      AND     Y5A6  ; U-BendInKnife UpSv
      SET     M6350  ; U-BendInKnife UpFlt
      MPP
      AND     Y5A7  ; U-BendInKnife DnSv
      SET     M6351  ; U-BendInKnife DnFlt
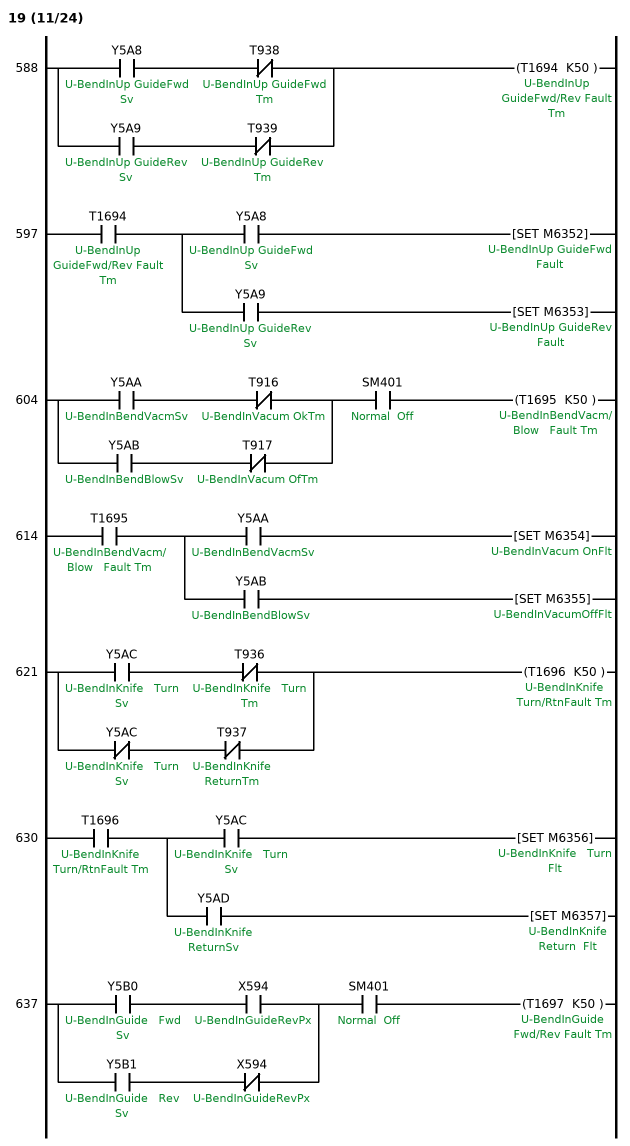
588   LD      Y5A8  ; U-BendInUp GuideFwd Sv
      ANI     T938  ; U-BendInUp GuideFwd Tm
      LD      Y5A9  ; U-BendInUp GuideRev Sv
      ANI     T939  ; U-BendInUp GuideRev Tm
      ORB
      OUT     T1694 K50  ; U-BendInUp GuideFwd/Rev Fault Tm
597   LD      T1694  ; U-BendInUp GuideFwd/Rev Fault Tm
      MPS
      AND     Y5A8  ; U-BendInUp GuideFwd Sv
      SET     M6352  ; U-BendInUp GuideFwd     Fault
      MPP
      AND     Y5A9  ; U-BendInUp GuideRev Sv
      SET     M6353  ; U-BendInUp GuideRev     Fault
604   LD      Y5AA  ; U-BendInBendVacmSv
      ANI     T916  ; U-BendInVacum OkTm
      LD      Y5AB  ; U-BendInBendBlowSv
      ANI     T917  ; U-BendInVacum OfTm
      ORB
      AND     SM401  ; Normal  Off
      OUT     T1695 K50  ; U-BendInBendVacm/Blow   Fault Tm
614   LD      T1695  ; U-BendInBendVacm/Blow   Fault Tm
      MPS
      AND     Y5AA  ; U-BendInBendVacmSv
      SET     M6354  ; U-BendInVacum OnFlt
      MPP
      AND     Y5AB  ; U-BendInBendBlowSv
      SET     M6355  ; U-BendInVacumOffFlt
621   LD      Y5AC  ; U-BendInKnife   Turn Sv
      ANI     T936  ; U-BendInKnife   Turn Tm
      LDI     Y5AC  ; U-BendInKnife   Turn Sv
      ANI     T937  ; U-BendInKnife   ReturnTm
      ORB
      OUT     T1696 K50  ; U-BendInKnife   Turn/RtnFault Tm
630   LD      T1696  ; U-BendInKnife   Turn/RtnFault Tm
      MPS
      AND     Y5AC  ; U-BendInKnife   Turn Sv
      SET     M6356  ; U-BendInKnife   Turn Flt
      MPP
      AND     Y5AD  ; U-BendInKnife   ReturnSv
      SET     M6357  ; U-BendInKnife   Return  Flt
637   LD      Y5B0  ; U-BendInGuide   Fwd Sv
      AND     X594  ; U-BendInGuideRevPx
      LD      Y5B1  ; U-BendInGuide   Rev Sv
      ANI     X594  ; U-BendInGuideRevPx
      ORB
      AND     SM401  ; Normal  Off
      OUT     T1697 K50  ; U-BendInGuide   Fwd/Rev Fault Tm
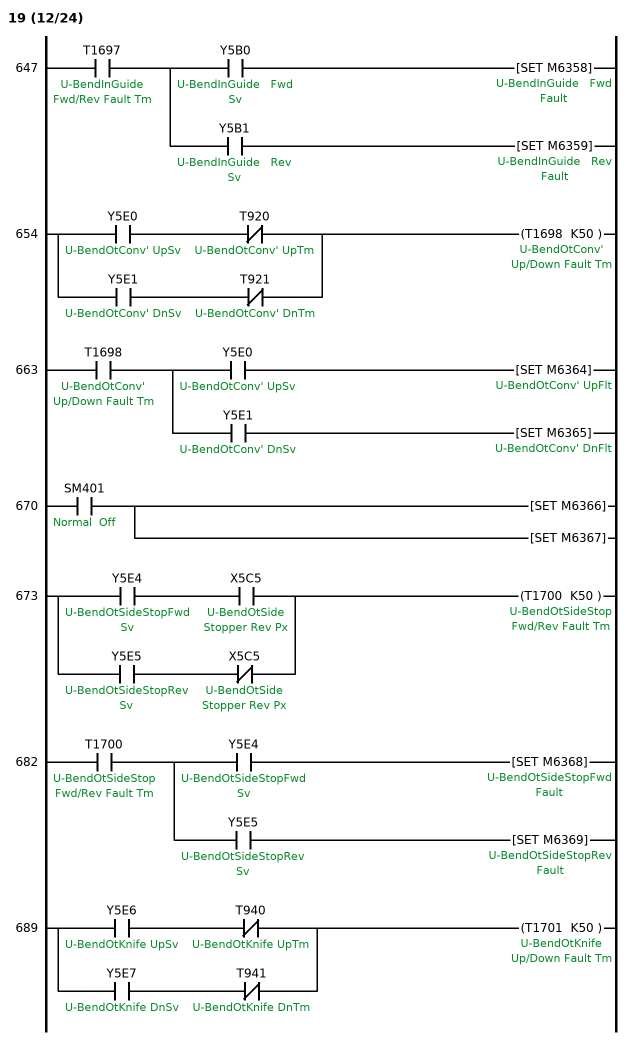
647   LD      T1697  ; U-BendInGuide   Fwd/Rev Fault Tm
      MPS
      AND     Y5B0  ; U-BendInGuide   Fwd Sv
      SET     M6358  ; U-BendInGuide   Fwd     Fault
      MPP
      AND     Y5B1  ; U-BendInGuide   Rev Sv
      SET     M6359  ; U-BendInGuide   Rev     Fault
654   LD      Y5E0  ; U-BendOtConv' UpSv
      ANI     T920  ; U-BendOtConv' UpTm
      LD      Y5E1  ; U-BendOtConv' DnSv
      ANI     T921  ; U-BendOtConv' DnTm
      ORB
      OUT     T1698 K50  ; U-BendOtConv'   Up/Down Fault Tm
663   LD      T1698  ; U-BendOtConv'   Up/Down Fault Tm
      MPS
      AND     Y5E0  ; U-BendOtConv' UpSv
      SET     M6364  ; U-BendOtConv' UpFlt
      MPP
      AND     Y5E1  ; U-BendOtConv' DnSv
      SET     M6365  ; U-BendOtConv' DnFlt
670   LD      SM401  ; Normal  Off
      SET     M6366
      SET     M6367
673   LD      Y5E4  ; U-BendOtSideStopFwd     Sv
      AND     X5C5  ; U-BendOtSide    Stopper Rev Px
      LD      Y5E5  ; U-BendOtSideStopRev     Sv
      ANI     X5C5  ; U-BendOtSide    Stopper Rev Px
      ORB
      OUT     T1700 K50  ; U-BendOtSideStopFwd/Rev Fault Tm
682   LD      T1700  ; U-BendOtSideStopFwd/Rev Fault Tm
      MPS
      AND     Y5E4  ; U-BendOtSideStopFwd     Sv
      SET     M6368  ; U-BendOtSideStopFwd     Fault
      MPP
      AND     Y5E5  ; U-BendOtSideStopRev     Sv
      SET     M6369  ; U-BendOtSideStopRev     Fault
689   LD      Y5E6  ; U-BendOtKnife UpSv
      ANI     T940  ; U-BendOtKnife UpTm
      LD      Y5E7  ; U-BendOtKnife DnSv
      ANI     T941  ; U-BendOtKnife DnTm
      ORB
      OUT     T1701 K50  ; U-BendOtKnife   Up/Down Fault Tm
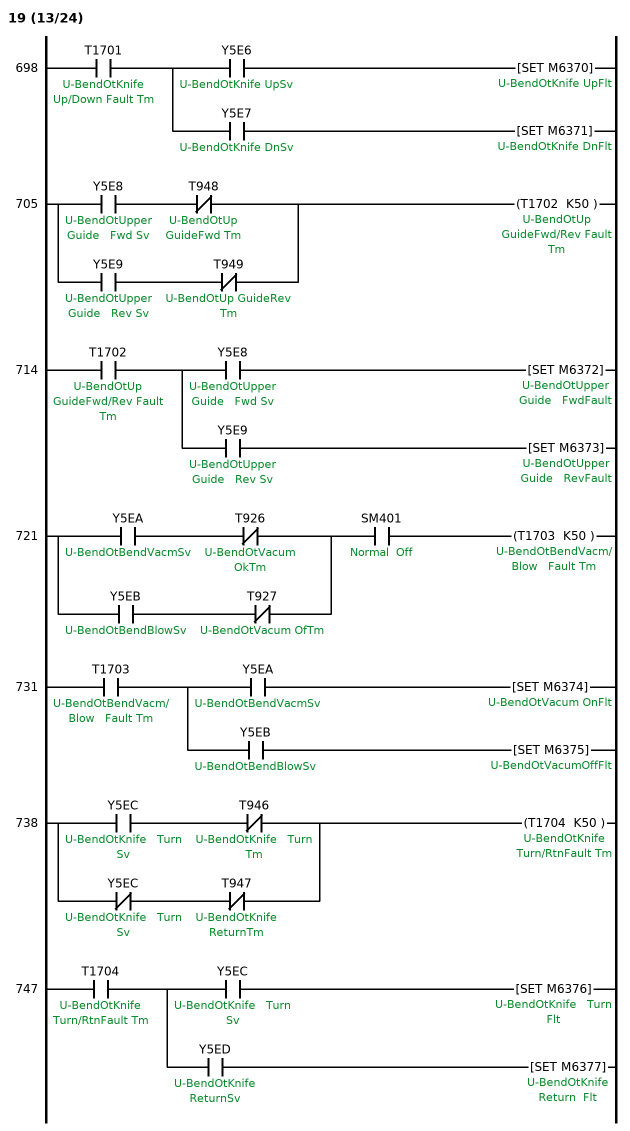
698   LD      T1701  ; U-BendOtKnife   Up/Down Fault Tm
      MPS
      AND     Y5E6  ; U-BendOtKnife UpSv
      SET     M6370  ; U-BendOtKnife UpFlt
      MPP
      AND     Y5E7  ; U-BendOtKnife DnSv
      SET     M6371  ; U-BendOtKnife DnFlt
705   LD      Y5E8  ; U-BendOtUpper   Guide   Fwd Sv
      ANI     T948  ; U-BendOtUp GuideFwd Tm
      LD      Y5E9  ; U-BendOtUpper   Guide   Rev Sv
      ANI     T949  ; U-BendOtUp GuideRev Tm
      ORB
      OUT     T1702 K50  ; U-BendOtUp GuideFwd/Rev Fault Tm
714   LD      T1702  ; U-BendOtUp GuideFwd/Rev Fault Tm
      MPS
      AND     Y5E8  ; U-BendOtUpper   Guide   Fwd Sv
      SET     M6372  ; U-BendOtUpper   Guide   FwdFault
      MPP
      AND     Y5E9  ; U-BendOtUpper   Guide   Rev Sv
      SET     M6373  ; U-BendOtUpper   Guide   RevFault
721   LD      Y5EA  ; U-BendOtBendVacmSv
      ANI     T926  ; U-BendOtVacum OkTm
      LD      Y5EB  ; U-BendOtBendBlowSv
      ANI     T927  ; U-BendOtVacum OfTm
      ORB
      AND     SM401  ; Normal  Off
      OUT     T1703 K50  ; U-BendOtBendVacm/Blow   Fault Tm
731   LD      T1703  ; U-BendOtBendVacm/Blow   Fault Tm
      MPS
      AND     Y5EA  ; U-BendOtBendVacmSv
      SET     M6374  ; U-BendOtVacum OnFlt
      MPP
      AND     Y5EB  ; U-BendOtBendBlowSv
      SET     M6375  ; U-BendOtVacumOffFlt
738   LD      Y5EC  ; U-BendOtKnife   Turn Sv
      ANI     T946  ; U-BendOtKnife   Turn Tm
      LDI     Y5EC  ; U-BendOtKnife   Turn Sv
      ANI     T947  ; U-BendOtKnife   ReturnTm
      ORB
      OUT     T1704 K50  ; U-BendOtKnife   Turn/RtnFault Tm
747   LD      T1704  ; U-BendOtKnife   Turn/RtnFault Tm
      MPS
      AND     Y5EC  ; U-BendOtKnife   Turn Sv
      SET     M6376  ; U-BendOtKnife   Turn Flt
      MPP
      AND     Y5ED  ; U-BendOtKnife   ReturnSv
      SET     M6377  ; U-BendOtKnife   Return  Flt
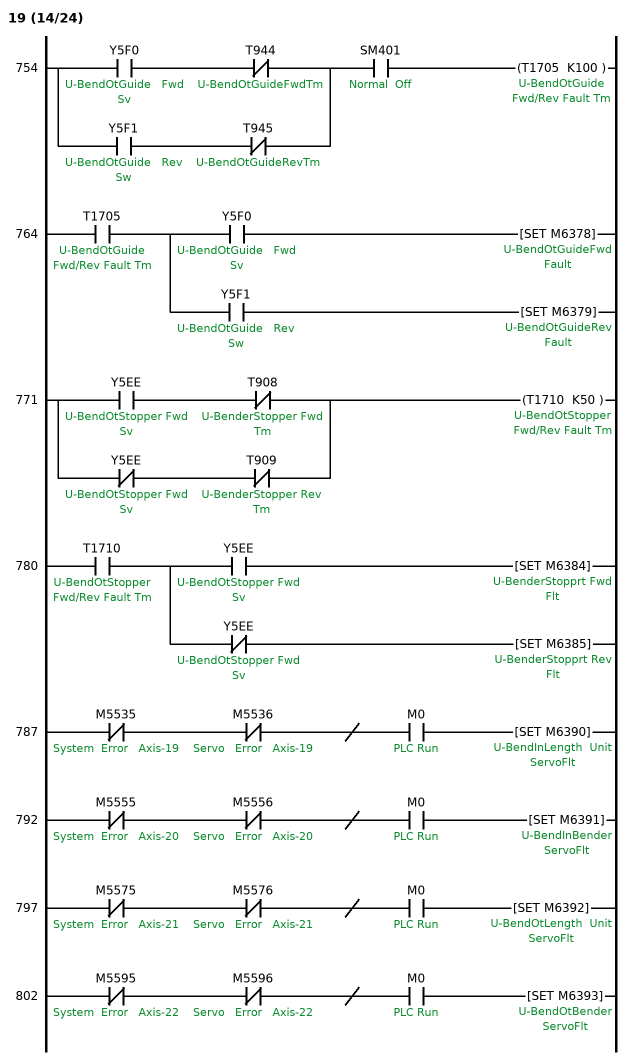
754   LD      Y5F0  ; U-BendOtGuide   Fwd Sv
      ANI     T944  ; U-BendOtGuideFwdTm
      LD      Y5F1  ; U-BendOtGuide   Rev Sw
      ANI     T945  ; U-BendOtGuideRevTm
      ORB
      AND     SM401  ; Normal  Off
      OUT     T1705 K100  ; U-BendOtGuide   Fwd/Rev Fault Tm
764   LD      T1705  ; U-BendOtGuide   Fwd/Rev Fault Tm
      MPS
      AND     Y5F0  ; U-BendOtGuide   Fwd Sv
      SET     M6378  ; U-BendOtGuideFwdFault
      MPP
      AND     Y5F1  ; U-BendOtGuide   Rev Sw
      SET     M6379  ; U-BendOtGuideRevFault
771   LD      Y5EE  ; U-BendOtStopper Fwd Sv
      ANI     T908  ; U-BenderStopper Fwd Tm
      LDI     Y5EE  ; U-BendOtStopper Fwd Sv
      ANI     T909  ; U-BenderStopper Rev Tm
      ORB
      OUT     T1710 K50  ; U-BendOtStopper Fwd/Rev Fault Tm
780   LD      T1710  ; U-BendOtStopper Fwd/Rev Fault Tm
      MPS
      AND     Y5EE  ; U-BendOtStopper Fwd Sv
      SET     M6384  ; U-BenderStopprt Fwd Flt
      MPP
      ANI     Y5EE  ; U-BendOtStopper Fwd Sv
      SET     M6385  ; U-BenderStopprt Rev Flt
787   LDI     M5535  ; System  Error   Axis-19
      ANI     M5536  ; Servo   Error   Axis-19
      INV
      AND     M0  ; PLC Run
      SET     M6390  ; U-BendInLength  Unit    ServoFlt
792   LDI     M5555  ; System  Error   Axis-20
      ANI     M5556  ; Servo   Error   Axis-20
      INV
      AND     M0  ; PLC Run
      SET     M6391  ; U-BendInBender  ServoFlt
797   LDI     M5575  ; System  Error   Axis-21
      ANI     M5576  ; Servo   Error   Axis-21
      INV
      AND     M0  ; PLC Run
      SET     M6392  ; U-BendOtLength  Unit    ServoFlt
802   LDI     M5595  ; System  Error   Axis-22
      ANI     M5596  ; Servo   Error   Axis-22
      INV
      AND     M0  ; PLC Run
      SET     M6393  ; U-BendOtBender  ServoFlt
